SPLINE
SPL {X  -133.736, Y  +773.248, Z    +0.000, E1   -45.385, E3 +353303.340}
SPL {X  -160.761, Y  +715.447, Z    +0.000, E1   -23.748, E3 +353260.190}
SPL {X  -164.304, Y  +696.571, Z    +0.000, E1   -14.525, E3 +353265.413}
SPL {X  -165.498, Y  +682.585, Z    +0.000, E1    -6.769, E3 +353265.088}
SPL {X  -165.650, Y  +674.975, Z    +0.000, E1    -1.888, E3 +353263.446}
SPL {X  -165.650, Y  +671.520, Z    +0.000, E1    +0.682, E3 +353262.373}
SPL {X  -165.650, Y  +668.289, Z    +0.000, E1    +3.417, E3 +353262.215}
SPL {X  -165.650, Y  +663.040, Z    +0.000, E1    +8.602, E3 +353261.410}
SPL {X  -165.650, Y  +655.692, Z    +0.000, E1   +17.061, E3 +353259.945}
SPL {X  -165.650, Y  +646.511, Z    +0.000, E1   +26.434, E3 +353262.725}
SPL {X  -165.650, Y  +637.905, Z    +0.000, E1   +40.225, E3 +353250.850}
SPL {X  -165.650, Y  +611.479, Z    +0.000, E1   +52.226, E3 +353264.402}
SPL {X  -165.650, Y  +599.923, Z    +0.000, E1   +51.240, E3 +353281.492}
SPL {X  -165.650, Y  +553.219, Z    +0.000, E1   +52.865, E3 +353338.252}
ENDSPLINE

SPLINE
SPL {X  -165.650, Y  +569.883, Z    +0.000, E1   +45.183, E3 +353353.929}
ENDSPLINE

SPLINE
SPL {X  -165.650, Y  +561.960, Z    +0.000, E1   +45.285, E3 +353369.584}
SPL {X  -165.650, Y  +554.065, Z    +0.000, E1   +45.254, E3 +353385.646}
SPL {X  -165.650, Y  +548.074, Z    +0.000, E1   +45.245, E3 +353397.757}
SPL {X  -165.650, Y  +542.958, Z    +0.000, E1   +45.131, E3 +353408.888}
SPL {X  -165.650, Y  +535.288, Z    +0.000, E1   +45.332, E3 +353423.328}
SPL {X  -165.650, Y  +529.160, Z    +0.000, E1   +45.215, E3 +353436.309}
SPL {X  -165.650, Y  +522.672, Z    +0.000, E1   +45.331, E3 +353448.876}
SPL {X  -165.650, Y  +516.211, Z    +0.000, E1   +45.175, E3 +353462.835}
SPL {X  -165.650, Y  +509.762, Z    +0.000, E1   +45.191, E3 +353475.877}
SPL {X  -165.650, Y  +503.812, Z    +0.000, E1   +45.188, E3 +353487.916}
SPL {X  -165.650, Y  +499.646, Z    +0.000, E1   +44.886, E3 +353498.187}
ENDSPLINE

SPLINE
SPL {X  -165.650, Y  +514.834, Z    +0.000, E1   +36.829, E3 +353510.953}
ENDSPLINE

SPLINE
SPL {X  -165.650, Y  +506.421, Z    +0.000, E1   +37.886, E3 +353527.065}
SPL {X  -165.650, Y  +499.917, Z    +0.000, E1   +38.752, E3 +353538.526}
SPL {X  -165.650, Y  +493.826, Z    +0.000, E1   +39.521, E3 +353549.280}
SPL {X  -165.650, Y  +487.003, Z    +0.000, E1   +40.380, E3 +353560.734}
SPL {X  -165.650, Y  +478.382, Z    +0.000, E1   +41.628, E3 +353573.647}
SPL {X  -165.650, Y  +472.112, Z    +0.000, E1   +42.202, E3 +353584.386}
SPL {X  -165.650, Y  +466.741, Z    +0.000, E1   +42.890, E3 +353592.306}
SPL {X  -165.650, Y  +458.202, Z    +0.000, E1   +44.020, E3 +353604.094}
SPL {X  -165.650, Y  +449.099, Z    +0.000, E1   +44.871, E3 +353618.056}
SPL {X  -165.650, Y  +442.120, Z    +0.000, E1   +45.313, E3 +353629.608}
SPL {X  -165.650, Y  +436.063, Z    +0.000, E1   +44.972, E3 +353644.193}
SPL {X  -165.650, Y  +427.943, Z    +0.000, E1   +45.362, E3 +353658.230}
SPL {X  -165.650, Y  +422.523, Z    +0.000, E1   +45.103, E3 +353670.908}
SPL {X  -165.650, Y  +415.564, Z    +0.000, E1   +45.195, E3 +353684.447}
SPL {X  -165.650, Y  +410.687, Z    +0.000, E1   +44.955, E3 +353695.763}
SPL {X  -165.650, Y  +405.522, Z    +0.000, E1   +45.119, E3 +353705.324}
SPL {X  -165.650, Y  +399.216, Z    +0.000, E1   +45.246, E3 +353717.517}
SPL {X  -165.650, Y  +391.618, Z    +0.000, E1   +45.037, E3 +353734.296}
SPL {X  -165.650, Y  +383.700, Z    +0.000, E1   +45.345, E3 +353748.422}
SPL {X  -165.650, Y  +379.225, Z    +0.000, E1   +45.073, E3 +353759.111}
SPL {X  -165.591, Y  +374.097, Z    +0.000, E1   +45.069, E3 +353769.592}
SPL {X  -165.372, Y  +368.914, Z    +0.000, E1   +45.103, E3 +353779.952}
SPL {X  -164.987, Y  +363.696, Z    +0.000, E1   +45.006, E3 +353791.175}
SPL {X  -164.256, Y  +357.053, Z    +0.000, E1   +44.969, E3 +353804.978}
SPL {X  -163.441, Y  +351.538, Z    +0.000, E1   +44.749, E3 +353817.341}
SPL {X  -162.419, Y  +345.942, Z    +0.000, E1   +44.540, E3 +353830.073}
SPL {X  -161.210, Y  +340.404, Z    +0.000, E1   +44.250, E3 +353842.898}
SPL {X  -159.961, Y  +335.460, Z    +0.000, E1   +44.205, E3 +353853.261}
SPL {X  -158.595, Y  +330.672, Z    +0.000, E1   +43.797, E3 +353865.239}
SPL {X  -157.207, Y  +326.289, Z    +0.000, E1   +43.631, E3 +353874.992}
SPL {X  -152.192, Y  +313.097, Z    +0.000, E1   +47.715, E3 +353878.546}
SPL {X  -146.385, Y  +300.967, Z    +0.000, E1   +50.402, E3 +353884.741}
SPL {X  -137.641, Y  +286.333, Z    +0.000, E1   +45.396, E3 +353956.232}
SPL {X  -137.518, Y  +286.149, Z    +0.000, E1   +42.648, E3 +354028.741}
ENDSPLINE

SPLINE
SPL {X  -156.430, Y  +324.005, Z    +0.000, E1   +29.926, E3 +354033.876}
SPL {X  -161.387, Y  +341.161, Z    +0.000, E1   +22.590, E3 +354049.718}
SPL {X  -164.566, Y  +359.576, Z    +0.000, E1   +13.425, E3 +354028.311}
SPL {X  -165.355, Y  +368.611, Z    +0.000, E1    +8.407, E3 +354031.892}
SPL {X  -165.614, Y  +375.050, Z    +0.000, E1    +4.520, E3 +354033.196}
SPL {X  -165.650, Y  +379.847, Z    +0.000, E1    +1.364, E3 +354031.545}
SPL {X  -165.650, Y  +384.387, Z    +0.000, E1    -2.084, E3 +354030.527}
SPL {X  -165.650, Y  +387.977, Z    +0.000, E1    -5.454, E3 +354031.012}
SPL {X  -165.650, Y  +392.464, Z    +0.000, E1   -10.170, E3 +354028.695}
SPL {X  -165.650, Y  +397.361, Z    +0.000, E1   -15.736, E3 +354028.027}
SPL {X  -165.650, Y  +404.553, Z    +0.000, E1   -23.488, E3 +354028.803}
SPL {X  -165.650, Y  +415.773, Z    +0.000, E1   -36.308, E3 +354024.955}
SPL {X  -165.650, Y  +461.620, Z    +0.000, E1   -55.594, E3 +354044.685}
SPL {X  -165.650, Y  +498.574, Z    +0.000, E1   -52.082, E3 +354105.710}
ENDSPLINE

SPLINE
SPL {X  -165.650, Y  +484.983, Z    +0.000, E1   -45.406, E3 +354121.213}
ENDSPLINE

SPLINE
SPL {X  -165.650, Y  +492.090, Z    +0.000, E1   -45.292, E3 +354136.235}
SPL {X  -165.650, Y  +498.857, Z    +0.000, E1   -45.339, E3 +354149.572}
SPL {X  -165.650, Y  +505.115, Z    +0.000, E1   -45.299, E3 +354162.520}
SPL {X  -165.650, Y  +510.931, Z    +0.000, E1   -45.250, E3 +354174.511}
SPL {X  -165.650, Y  +516.157, Z    +0.000, E1   -45.240, E3 +354185.186}
SPL {X  -165.650, Y  +521.049, Z    +0.000, E1   -45.236, E3 +354195.138}
SPL {X  -165.650, Y  +527.050, Z    +0.000, E1   -45.345, E3 +354206.634}
SPL {X  -165.650, Y  +532.042, Z    +0.000, E1   -45.233, E3 +354217.378}
SPL {X  -165.650, Y  +537.290, Z    +0.000, E1   -45.204, E3 +354228.219}
SPL {X  -165.650, Y  +544.196, Z    +0.000, E1   -45.432, E3 +354240.893}
SPL {X  -165.650, Y  +548.678, Z    +0.000, E1   -45.162, E3 +354251.457}
SPL {X  -165.650, Y  +554.600, Z    +0.000, E1   -45.345, E3 +354262.434}
SPL {X  -165.650, Y  +559.896, Z    +0.000, E1   -45.150, E3 +354274.289}
SPL {X  -165.650, Y  +566.830, Z    +0.000, E1   -45.346, E3 +354287.269}
SPL {X  -165.650, Y  +573.074, Z    +0.000, E1   -45.379, E3 +354299.600}
SPL {X  -165.650, Y  +579.360, Z    +0.000, E1   -45.300, E3 +354312.885}
SPL {X  -165.650, Y  +584.577, Z    +0.000, E1   -45.167, E3 +354324.108}
SPL {X  -165.650, Y  +590.060, Z    +0.000, E1   -45.221, E3 +354334.999}
SPL {X  -165.650, Y  +596.611, Z    +0.000, E1   -45.390, E3 +354347.236}
SPL {X  -165.650, Y  +603.637, Z    +0.000, E1   -45.296, E3 +354362.154}
SPL {X  -165.650, Y  +610.850, Z    +0.000, E1   -45.208, E3 +354377.162}
SPL {X  -165.650, Y  +617.450, Z    +0.000, E1   -45.402, E3 +354389.365}
SPL {X  -165.650, Y  +622.720, Z    +0.000, E1   -45.272, E3 +354400.763}
SPL {X  -165.650, Y  +627.828, Z    +0.000, E1   -45.174, E3 +354411.719}
SPL {X  -165.650, Y  +634.620, Z    +0.000, E1   -45.438, E3 +354423.925}
SPL {X  -165.650, Y  +640.808, Z    +0.000, E1   -45.294, E3 +354437.299}
SPL {X  -165.650, Y  +646.552, Z    +0.000, E1   -45.137, E3 +354449.824}
SPL {X  -165.650, Y  +652.431, Z    +0.000, E1   -45.333, E3 +354460.578}
SPL {X  -165.650, Y  +657.443, Z    +0.000, E1   -45.316, E3 +354470.834}
SPL {X  -165.650, Y  +662.999, Z    +0.000, E1   -45.214, E3 +354482.706}
SPL {X  -165.650, Y  +668.737, Z    +0.000, E1   -45.236, E3 +354494.221}
SPL {X  -165.650, Y  +675.226, Z    +0.000, E1   -45.503, E3 +354505.725}
SPL {X  -165.597, Y  +679.672, Z    +0.000, E1   -45.206, E3 +354516.446}
SPL {X  -165.388, Y  +684.808, Z    +0.000, E1   -45.192, E3 +354526.954}
SPL {X  -165.020, Y  +689.938, Z    +0.000, E1   -45.107, E3 +354537.896}
SPL {X  -164.358, Y  +696.147, Z    +0.000, E1   -45.160, E3 +354550.162}
SPL {X  -163.631, Y  +701.286, Z    +0.000, E1   -44.994, E3 +354561.454}
SPL {X  -162.679, Y  +706.734, Z    +0.000, E1   -44.812, E3 +354573.687}
SPL {X  -161.655, Y  +711.661, Z    +0.000, E1   -44.525, E3 +354585.068}
SPL {X  -160.692, Y  +715.726, Z    +0.000, E1   -44.379, E3 +354594.225}
SPL {X  -159.384, Y  +720.631, Z    +0.000, E1   -44.155, E3 +354605.376}
SPL {X  -158.321, Y  +724.227, Z    +0.000, E1   -43.955, E3 +354613.697}
SPL {X  -156.604, Y  +729.490, Z    +0.000, E1   -44.229, E3 +354622.863}
SPL {X  -147.100, Y  +751.668, Z    +0.000, E1   -50.624, E3 +354628.750}
SPL {X  -144.116, Y  +757.172, Z    +0.000, E1   -42.809, E3 +354698.146}
SPL {X  -127.227, Y  +781.582, Z    +0.000, E1   -46.780, E3 +354743.816}
ENDSPLINE

SPLINE
SPL {X  -133.736, Y  +773.248, Z    +0.000, E1   -45.385, E3 +354821.858}
SPL {X  -160.761, Y  +715.447, Z    +0.000, E1   -23.748, E3 +354778.708}
SPL {X  -164.304, Y  +696.571, Z    +0.000, E1   -14.525, E3 +354783.932}
SPL {X  -165.498, Y  +682.585, Z    +0.000, E1    -6.769, E3 +354783.606}
SPL {X  -165.650, Y  +674.975, Z    +0.000, E1    -1.888, E3 +354781.965}
SPL {X  -165.650, Y  +671.520, Z    +0.000, E1    +0.682, E3 +354780.892}
SPL {X  -165.650, Y  +668.289, Z    +0.000, E1    +3.417, E3 +354780.734}
SPL {X  -165.650, Y  +663.040, Z    +0.000, E1    +8.602, E3 +354779.928}
SPL {X  -165.650, Y  +655.692, Z    +0.000, E1   +17.061, E3 +354778.464}
SPL {X  -165.650, Y  +646.511, Z    +0.000, E1   +26.434, E3 +354781.244}
SPL {X  -165.650, Y  +637.905, Z    +0.000, E1   +40.225, E3 +354769.368}
SPL {X  -165.650, Y  +611.479, Z    +0.000, E1   +52.226, E3 +354782.921}
SPL {X  -165.650, Y  +599.923, Z    +0.000, E1   +51.240, E3 +354800.010}
SPL {X  -165.650, Y  +553.219, Z    +0.000, E1   +52.865, E3 +354856.771}
ENDSPLINE

SPLINE
SPL {X  -165.650, Y  +569.883, Z    +0.000, E1   +45.183, E3 +354872.447}
ENDSPLINE

SPLINE
SPL {X  -165.650, Y  +561.960, Z    +0.000, E1   +45.285, E3 +354888.103}
SPL {X  -165.650, Y  +554.065, Z    +0.000, E1   +45.254, E3 +354904.165}
SPL {X  -165.650, Y  +548.074, Z    +0.000, E1   +45.245, E3 +354916.275}
SPL {X  -165.650, Y  +542.958, Z    +0.000, E1   +45.131, E3 +354927.406}
SPL {X  -165.650, Y  +535.288, Z    +0.000, E1   +45.332, E3 +354941.847}
SPL {X  -165.650, Y  +529.160, Z    +0.000, E1   +45.215, E3 +354954.828}
SPL {X  -165.650, Y  +522.672, Z    +0.000, E1   +45.331, E3 +354967.394}
SPL {X  -165.650, Y  +516.211, Z    +0.000, E1   +45.175, E3 +354981.354}
SPL {X  -165.650, Y  +509.762, Z    +0.000, E1   +45.191, E3 +354994.396}
SPL {X  -165.650, Y  +503.812, Z    +0.000, E1   +45.188, E3 +355006.434}
SPL {X  -165.650, Y  +499.646, Z    +0.000, E1   +44.886, E3 +355016.705}
ENDSPLINE

SPLINE
SPL {X  -165.650, Y  +516.930, Z    +0.000, E1   +36.544, E3 +355025.376}
ENDSPLINE

SPLINE
SPL {X  -165.650, Y  +511.324, Z    +0.000, E1   +37.254, E3 +355036.367}
SPL {X  -165.650, Y  +504.742, Z    +0.000, E1   +38.087, E3 +355048.672}
SPL {X  -165.650, Y  +497.845, Z    +0.000, E1   +39.022, E3 +355060.747}
SPL {X  -165.650, Y  +491.819, Z    +0.000, E1   +39.756, E3 +355071.266}
SPL {X  -165.650, Y  +485.086, Z    +0.000, E1   +40.678, E3 +355082.110}
SPL {X  -165.650, Y  +476.633, Z    +0.000, E1   +41.847, E3 +355094.809}
SPL {X  -165.650, Y  +468.596, Z    +0.000, E1   +42.673, E3 +355108.072}
SPL {X  -165.650, Y  +460.562, Z    +0.000, E1   +43.733, E3 +355119.224}
SPL {X  -165.650, Y  +455.629, Z    +0.000, E1   +44.293, E3 +355126.343}
SPL {X  -165.650, Y  +449.099, Z    +0.000, E1   +44.871, E3 +355136.575}
SPL {X  -165.650, Y  +442.120, Z    +0.000, E1   +45.313, E3 +355148.127}
SPL {X  -165.650, Y  +439.103, Z    +0.000, E1   +44.726, E3 +355157.736}
SPL {X  -165.650, Y  +433.421, Z    +0.000, E1   +45.110, E3 +355167.123}
SPL {X  -165.650, Y  +426.476, Z    +0.000, E1   +45.244, E3 +355180.627}
SPL {X  -165.650, Y  +420.418, Z    +0.000, E1   +45.128, E3 +355193.421}
SPL {X  -165.650, Y  +415.564, Z    +0.000, E1   +45.195, E3 +355202.966}
SPL {X  -165.650, Y  +410.687, Z    +0.000, E1   +44.955, E3 +355214.282}
SPL {X  -165.650, Y  +405.522, Z    +0.000, E1   +45.119, E3 +355223.842}
SPL {X  -165.650, Y  +400.300, Z    +0.000, E1   +45.439, E3 +355232.526}
SPL {X  -165.650, Y  +396.171, Z    +0.000, E1   +44.969, E3 +355243.783}
SPL {X  -165.650, Y  +390.060, Z    +0.000, E1   +45.007, E3 +355256.017}
SPL {X  -165.650, Y  +383.700, Z    +0.000, E1   +45.345, E3 +355266.941}
SPL {X  -165.650, Y  +379.225, Z    +0.000, E1   +45.073, E3 +355277.630}
SPL {X  -165.591, Y  +374.097, Z    +0.000, E1   +45.069, E3 +355288.111}
SPL {X  -165.372, Y  +368.914, Z    +0.000, E1   +45.103, E3 +355298.471}
SPL {X  -164.987, Y  +363.696, Z    +0.000, E1   +45.006, E3 +355309.694}
SPL {X  -164.256, Y  +357.053, Z    +0.000, E1   +44.969, E3 +355323.496}
SPL {X  -163.441, Y  +351.538, Z    +0.000, E1   +44.749, E3 +355335.860}
SPL {X  -162.419, Y  +345.942, Z    +0.000, E1   +44.540, E3 +355348.592}
SPL {X  -161.210, Y  +340.404, Z    +0.000, E1   +44.250, E3 +355361.417}
SPL {X  -159.961, Y  +335.460, Z    +0.000, E1   +44.205, E3 +355371.779}
SPL {X  -158.595, Y  +330.672, Z    +0.000, E1   +43.797, E3 +355383.758}
SPL {X  -157.207, Y  +326.289, Z    +0.000, E1   +43.631, E3 +355393.511}
SPL {X  -152.192, Y  +313.097, Z    +0.000, E1   +47.715, E3 +355397.064}
SPL {X  -146.385, Y  +300.967, Z    +0.000, E1   +50.402, E3 +355403.260}
SPL {X  -138.435, Y  +287.529, Z    +0.000, E1   +45.834, E3 +355465.216}
SPL {X  -134.645, Y  +282.008, Z    +0.000, E1   +45.207, E3 +355494.872}
ENDSPLINE

SPLINE
SPL {X  -154.915, Y  +319.839, Z    +0.000, E1   +31.584, E3 +355554.391}
SPL {X  -161.387, Y  +341.161, Z    +0.000, E1   +22.590, E3 +355568.236}
SPL {X  -164.566, Y  +359.576, Z    +0.000, E1   +13.425, E3 +355546.830}
SPL {X  -165.355, Y  +368.611, Z    +0.000, E1    +8.407, E3 +355550.411}
SPL {X  -165.614, Y  +375.050, Z    +0.000, E1    +4.520, E3 +355551.714}
SPL {X  -165.650, Y  +379.847, Z    +0.000, E1    +1.364, E3 +355550.064}
SPL {X  -165.650, Y  +383.246, Z    +0.000, E1    -1.216, E3 +355549.157}
SPL {X  -165.650, Y  +386.866, Z    +0.000, E1    -4.337, E3 +355549.210}
SPL {X  -165.650, Y  +392.464, Z    +0.000, E1   -10.170, E3 +355547.213}
SPL {X  -165.650, Y  +397.361, Z    +0.000, E1   -15.736, E3 +355546.545}
SPL {X  -165.650, Y  +404.553, Z    +0.000, E1   -23.488, E3 +355547.321}
SPL {X  -165.650, Y  +415.773, Z    +0.000, E1   -36.308, E3 +355543.474}
SPL {X  -165.650, Y  +456.525, Z    +0.000, E1   -55.091, E3 +355559.036}
SPL {X  -165.650, Y  +467.178, Z    +0.000, E1   -56.049, E3 +355567.773}
SPL {X  -165.650, Y  +498.574, Z    +0.000, E1   -52.082, E3 +355624.228}
ENDSPLINE

SPLINE
SPL {X  -165.650, Y  +484.983, Z    +0.000, E1   -45.406, E3 +355639.731}
ENDSPLINE

SPLINE
SPL {X  -165.650, Y  +492.090, Z    +0.000, E1   -45.292, E3 +355654.754}
SPL {X  -165.650, Y  +498.857, Z    +0.000, E1   -45.339, E3 +355668.091}
SPL {X  -165.650, Y  +504.159, Z    +0.000, E1   -45.384, E3 +355678.485}
SPL {X  -165.650, Y  +509.628, Z    +0.000, E1   -45.217, E3 +355690.669}
SPL {X  -165.650, Y  +516.157, Z    +0.000, E1   -45.240, E3 +355703.704}
SPL {X  -165.650, Y  +521.049, Z    +0.000, E1   -45.236, E3 +355713.657}
SPL {X  -165.650, Y  +527.050, Z    +0.000, E1   -45.345, E3 +355725.153}
SPL {X  -165.650, Y  +532.042, Z    +0.000, E1   -45.233, E3 +355735.896}
SPL {X  -165.650, Y  +537.290, Z    +0.000, E1   -45.204, E3 +355746.737}
SPL {X  -165.650, Y  +544.196, Z    +0.000, E1   -45.432, E3 +355759.411}
SPL {X  -165.650, Y  +548.678, Z    +0.000, E1   -45.162, E3 +355769.975}
SPL {X  -165.650, Y  +554.600, Z    +0.000, E1   -45.345, E3 +355780.952}
SPL {X  -165.650, Y  +561.799, Z    +0.000, E1   -45.312, E3 +355795.821}
SPL {X  -165.650, Y  +567.835, Z    +0.000, E1   -45.186, E3 +355808.628}
SPL {X  -165.650, Y  +573.074, Z    +0.000, E1   -45.379, E3 +355818.118}
SPL {X  -165.650, Y  +577.292, Z    +0.000, E1   -45.246, E3 +355827.382}
SPL {X  -165.650, Y  +583.131, Z    +0.000, E1   -45.255, E3 +355839.324}
SPL {X  -165.650, Y  +590.060, Z    +0.000, E1   -45.221, E3 +355853.518}
SPL {X  -165.650, Y  +596.611, Z    +0.000, E1   -45.390, E3 +355865.754}
SPL {X  -165.650, Y  +603.637, Z    +0.000, E1   -45.296, E3 +355880.673}
SPL {X  -165.650, Y  +610.850, Z    +0.000, E1   -45.208, E3 +355895.681}
SPL {X  -165.650, Y  +617.450, Z    +0.000, E1   -45.402, E3 +355907.883}
SPL {X  -165.650, Y  +622.720, Z    +0.000, E1   -45.272, E3 +355919.281}
SPL {X  -165.650, Y  +627.828, Z    +0.000, E1   -45.174, E3 +355930.238}
SPL {X  -165.650, Y  +634.620, Z    +0.000, E1   -45.438, E3 +355942.443}
SPL {X  -165.650, Y  +640.808, Z    +0.000, E1   -45.294, E3 +355955.818}
SPL {X  -165.650, Y  +646.552, Z    +0.000, E1   -45.137, E3 +355968.342}
SPL {X  -165.650, Y  +652.431, Z    +0.000, E1   -45.333, E3 +355979.097}
SPL {X  -165.650, Y  +657.443, Z    +0.000, E1   -45.316, E3 +355989.353}
SPL {X  -165.650, Y  +662.999, Z    +0.000, E1   -45.214, E3 +356001.225}
SPL {X  -165.650, Y  +668.737, Z    +0.000, E1   -45.236, E3 +356012.740}
SPL {X  -165.650, Y  +675.226, Z    +0.000, E1   -45.503, E3 +356024.243}
SPL {X  -165.597, Y  +679.672, Z    +0.000, E1   -45.206, E3 +356034.965}
SPL {X  -165.388, Y  +684.808, Z    +0.000, E1   -45.192, E3 +356045.472}
SPL {X  -165.020, Y  +689.938, Z    +0.000, E1   -45.107, E3 +356056.415}
SPL {X  -164.358, Y  +696.147, Z    +0.000, E1   -45.160, E3 +356068.681}
SPL {X  -163.631, Y  +701.286, Z    +0.000, E1   -44.994, E3 +356079.973}
SPL {X  -163.047, Y  +704.748, Z    +0.000, E1   -44.682, E3 +356088.796}
SPL {X  -161.884, Y  +710.619, Z    +0.000, E1   -44.738, E3 +356100.421}
SPL {X  -160.692, Y  +715.726, Z    +0.000, E1   -44.379, E3 +356112.744}
SPL {X  -158.938, Y  +722.175, Z    +0.000, E1   -44.121, E3 +356127.392}
SPL {X  -157.296, Y  +727.442, Z    +0.000, E1   -43.792, E3 +356139.617}
SPL {X  -153.030, Y  +738.918, Z    +0.000, E1   -47.123, E3 +356143.983}
SPL {X  -145.149, Y  +755.323, Z    +0.000, E1   -51.167, E3 +356150.115}
SPL {X  -143.038, Y  +759.047, Z    +0.000, E1   -43.157, E3 +356219.289}
SPL {X  -123.277, Y  +786.146, Z    +0.000, E1   -47.533, E3 +356275.344}
ENDSPLINE

SPLINE
SPL {X  -133.736, Y  +773.248, Z    +0.000, E1   -45.385, E3 +356340.377}
SPL {X  -160.761, Y  +715.447, Z    +0.000, E1   -23.748, E3 +356297.227}
SPL {X  -164.304, Y  +696.571, Z    +0.000, E1   -14.525, E3 +356302.451}
SPL {X  -165.498, Y  +682.585, Z    +0.000, E1    -6.769, E3 +356302.125}
SPL {X  -165.650, Y  +674.975, Z    +0.000, E1    -1.888, E3 +356300.483}
SPL {X  -165.650, Y  +671.520, Z    +0.000, E1    +0.682, E3 +356299.410}
SPL {X  -165.650, Y  +668.289, Z    +0.000, E1    +3.417, E3 +356299.252}
SPL {X  -165.650, Y  +663.040, Z    +0.000, E1    +8.602, E3 +356298.447}
SPL {X  -165.650, Y  +655.692, Z    +0.000, E1   +17.061, E3 +356296.982}
SPL {X  -165.650, Y  +646.511, Z    +0.000, E1   +26.434, E3 +356299.762}
SPL {X  -165.650, Y  +637.905, Z    +0.000, E1   +40.225, E3 +356287.887}
SPL {X  -165.650, Y  +611.479, Z    +0.000, E1   +52.226, E3 +356301.439}
SPL {X  -165.650, Y  +599.923, Z    +0.000, E1   +51.240, E3 +356318.529}
SPL {X  -165.650, Y  +553.219, Z    +0.000, E1   +52.865, E3 +356375.289}
ENDSPLINE

SPLINE
SPL {X  -165.650, Y  +569.883, Z    +0.000, E1   +45.183, E3 +356390.966}
ENDSPLINE

SPLINE
SPL {X  -165.650, Y  +561.960, Z    +0.000, E1   +45.285, E3 +356406.621}
SPL {X  -165.650, Y  +554.065, Z    +0.000, E1   +45.254, E3 +356422.683}
SPL {X  -165.650, Y  +548.074, Z    +0.000, E1   +45.245, E3 +356434.794}
SPL {X  -165.650, Y  +542.958, Z    +0.000, E1   +45.131, E3 +356445.925}
SPL {X  -165.650, Y  +535.288, Z    +0.000, E1   +45.332, E3 +356460.366}
SPL {X  -165.650, Y  +529.160, Z    +0.000, E1   +45.215, E3 +356473.346}
SPL {X  -165.650, Y  +522.672, Z    +0.000, E1   +45.331, E3 +356485.913}
SPL {X  -165.650, Y  +516.211, Z    +0.000, E1   +45.175, E3 +356499.872}
SPL {X  -165.650, Y  +509.762, Z    +0.000, E1   +45.191, E3 +356512.914}
SPL {X  -165.650, Y  +503.812, Z    +0.000, E1   +45.188, E3 +356524.953}
SPL {X  -165.650, Y  +499.646, Z    +0.000, E1   +44.886, E3 +356535.224}
ENDSPLINE

SPLINE
SPL {X  -165.650, Y  +514.834, Z    +0.000, E1   +36.829, E3 +356547.990}
ENDSPLINE

SPLINE
SPL {X  -165.650, Y  +506.421, Z    +0.000, E1   +37.886, E3 +356564.102}
SPL {X  -165.650, Y  +499.917, Z    +0.000, E1   +38.752, E3 +356575.563}
SPL {X  -165.650, Y  +493.826, Z    +0.000, E1   +39.521, E3 +356586.317}
SPL {X  -165.650, Y  +487.003, Z    +0.000, E1   +40.380, E3 +356597.771}
SPL {X  -165.650, Y  +478.382, Z    +0.000, E1   +41.628, E3 +356610.684}
SPL {X  -165.650, Y  +472.112, Z    +0.000, E1   +42.202, E3 +356621.423}
SPL {X  -165.650, Y  +466.741, Z    +0.000, E1   +42.890, E3 +356629.343}
SPL {X  -165.650, Y  +458.202, Z    +0.000, E1   +44.020, E3 +356641.131}
SPL {X  -165.650, Y  +449.099, Z    +0.000, E1   +44.871, E3 +356655.093}
SPL {X  -165.650, Y  +442.120, Z    +0.000, E1   +45.313, E3 +356666.645}
SPL {X  -165.650, Y  +436.063, Z    +0.000, E1   +44.972, E3 +356681.230}
SPL {X  -165.650, Y  +427.943, Z    +0.000, E1   +45.362, E3 +356695.267}
SPL {X  -165.650, Y  +422.523, Z    +0.000, E1   +45.103, E3 +356707.945}
SPL {X  -165.650, Y  +415.564, Z    +0.000, E1   +45.195, E3 +356721.484}
SPL {X  -165.650, Y  +410.687, Z    +0.000, E1   +44.955, E3 +356732.801}
SPL {X  -165.650, Y  +405.522, Z    +0.000, E1   +45.119, E3 +356742.361}
SPL {X  -165.650, Y  +399.216, Z    +0.000, E1   +45.246, E3 +356754.555}
SPL {X  -165.650, Y  +391.618, Z    +0.000, E1   +45.037, E3 +356771.333}
SPL {X  -165.650, Y  +383.700, Z    +0.000, E1   +45.345, E3 +356785.459}
SPL {X  -165.650, Y  +379.225, Z    +0.000, E1   +45.073, E3 +356796.148}
SPL {X  -165.591, Y  +374.097, Z    +0.000, E1   +45.069, E3 +356806.629}
SPL {X  -165.372, Y  +368.914, Z    +0.000, E1   +45.103, E3 +356816.989}
SPL {X  -164.987, Y  +363.696, Z    +0.000, E1   +45.006, E3 +356828.212}
SPL {X  -164.256, Y  +357.053, Z    +0.000, E1   +44.969, E3 +356842.015}
SPL {X  -163.441, Y  +351.538, Z    +0.000, E1   +44.749, E3 +356854.378}
SPL {X  -162.419, Y  +345.942, Z    +0.000, E1   +44.540, E3 +356867.110}
SPL {X  -161.210, Y  +340.404, Z    +0.000, E1   +44.250, E3 +356879.935}
SPL {X  -159.961, Y  +335.460, Z    +0.000, E1   +44.205, E3 +356890.298}
SPL {X  -158.595, Y  +330.672, Z    +0.000, E1   +43.797, E3 +356902.276}
SPL {X  -157.207, Y  +326.289, Z    +0.000, E1   +43.631, E3 +356912.029}
SPL {X  -152.192, Y  +313.097, Z    +0.000, E1   +47.715, E3 +356915.583}
SPL {X  -146.385, Y  +300.967, Z    +0.000, E1   +50.402, E3 +356921.778}
SPL {X  -137.641, Y  +286.333, Z    +0.000, E1   +45.396, E3 +356993.269}
SPL {X  -137.518, Y  +286.149, Z    +0.000, E1   +42.648, E3 +357065.779}
ENDSPLINE

SPLINE
SPL {X  -156.430, Y  +324.005, Z    +0.000, E1   +29.926, E3 +357070.913}
SPL {X  -161.387, Y  +341.161, Z    +0.000, E1   +22.590, E3 +357086.755}
SPL {X  -164.566, Y  +359.576, Z    +0.000, E1   +13.425, E3 +357065.348}
SPL {X  -165.355, Y  +368.611, Z    +0.000, E1    +8.407, E3 +357068.929}
SPL {X  -165.614, Y  +375.050, Z    +0.000, E1    +4.520, E3 +357070.233}
SPL {X  -165.650, Y  +379.847, Z    +0.000, E1    +1.364, E3 +357068.582}
SPL {X  -165.650, Y  +384.387, Z    +0.000, E1    -2.084, E3 +357067.564}
SPL {X  -165.650, Y  +387.977, Z    +0.000, E1    -5.454, E3 +357068.049}
SPL {X  -165.650, Y  +392.464, Z    +0.000, E1   -10.170, E3 +357065.732}
SPL {X  -165.650, Y  +397.361, Z    +0.000, E1   -15.736, E3 +357065.064}
SPL {X  -165.650, Y  +404.553, Z    +0.000, E1   -23.488, E3 +357065.840}
SPL {X  -165.650, Y  +415.773, Z    +0.000, E1   -36.308, E3 +357061.992}
SPL {X  -165.650, Y  +461.620, Z    +0.000, E1   -55.594, E3 +357081.722}
SPL {X  -165.650, Y  +498.574, Z    +0.000, E1   -52.082, E3 +357142.747}
ENDSPLINE

SPLINE
SPL {X  -165.650, Y  +484.983, Z    +0.000, E1   -45.406, E3 +357158.250}
ENDSPLINE

SPLINE
SPL {X  -165.650, Y  +492.090, Z    +0.000, E1   -45.292, E3 +357173.272}
SPL {X  -165.650, Y  +498.857, Z    +0.000, E1   -45.339, E3 +357186.609}
SPL {X  -165.650, Y  +505.115, Z    +0.000, E1   -45.299, E3 +357199.558}
SPL {X  -165.650, Y  +510.931, Z    +0.000, E1   -45.250, E3 +357211.548}
SPL {X  -165.650, Y  +516.157, Z    +0.000, E1   -45.240, E3 +357222.223}
SPL {X  -165.650, Y  +521.049, Z    +0.000, E1   -45.236, E3 +357232.175}
SPL {X  -165.650, Y  +527.050, Z    +0.000, E1   -45.345, E3 +357243.671}
SPL {X  -165.650, Y  +532.042, Z    +0.000, E1   -45.233, E3 +357254.415}
SPL {X  -165.650, Y  +537.290, Z    +0.000, E1   -45.204, E3 +357265.256}
SPL {X  -165.650, Y  +544.196, Z    +0.000, E1   -45.432, E3 +357277.930}
SPL {X  -165.650, Y  +548.678, Z    +0.000, E1   -45.162, E3 +357288.494}
SPL {X  -165.650, Y  +554.600, Z    +0.000, E1   -45.345, E3 +357299.471}
SPL {X  -165.650, Y  +559.896, Z    +0.000, E1   -45.150, E3 +357311.326}
SPL {X  -165.650, Y  +566.830, Z    +0.000, E1   -45.346, E3 +357324.306}
SPL {X  -165.650, Y  +573.074, Z    +0.000, E1   -45.379, E3 +357336.637}
SPL {X  -165.650, Y  +579.360, Z    +0.000, E1   -45.300, E3 +357349.922}
SPL {X  -165.650, Y  +584.577, Z    +0.000, E1   -45.167, E3 +357361.145}
SPL {X  -165.650, Y  +590.060, Z    +0.000, E1   -45.221, E3 +357372.036}
SPL {X  -165.650, Y  +596.611, Z    +0.000, E1   -45.390, E3 +357384.273}
SPL {X  -165.650, Y  +603.637, Z    +0.000, E1   -45.296, E3 +357399.191}
SPL {X  -165.650, Y  +610.850, Z    +0.000, E1   -45.208, E3 +357414.199}
SPL {X  -165.650, Y  +617.450, Z    +0.000, E1   -45.402, E3 +357426.402}
SPL {X  -165.650, Y  +622.720, Z    +0.000, E1   -45.272, E3 +357437.800}
SPL {X  -165.650, Y  +627.828, Z    +0.000, E1   -45.174, E3 +357448.756}
SPL {X  -165.650, Y  +634.620, Z    +0.000, E1   -45.438, E3 +357460.962}
SPL {X  -165.650, Y  +640.808, Z    +0.000, E1   -45.294, E3 +357474.336}
SPL {X  -165.650, Y  +646.552, Z    +0.000, E1   -45.137, E3 +357486.861}
SPL {X  -165.650, Y  +652.431, Z    +0.000, E1   -45.333, E3 +357497.615}
SPL {X  -165.650, Y  +657.443, Z    +0.000, E1   -45.316, E3 +357507.871}
SPL {X  -165.650, Y  +662.999, Z    +0.000, E1   -45.214, E3 +357519.743}
SPL {X  -165.650, Y  +668.737, Z    +0.000, E1   -45.236, E3 +357531.258}
SPL {X  -165.650, Y  +675.226, Z    +0.000, E1   -45.503, E3 +357542.762}
SPL {X  -165.597, Y  +679.672, Z    +0.000, E1   -45.206, E3 +357553.483}
SPL {X  -165.388, Y  +684.808, Z    +0.000, E1   -45.192, E3 +357563.991}
SPL {X  -165.020, Y  +689.938, Z    +0.000, E1   -45.107, E3 +357574.933}
SPL {X  -164.358, Y  +696.147, Z    +0.000, E1   -45.160, E3 +357587.199}
SPL {X  -163.631, Y  +701.286, Z    +0.000, E1   -44.994, E3 +357598.491}
SPL {X  -162.679, Y  +706.734, Z    +0.000, E1   -44.812, E3 +357610.724}
SPL {X  -161.655, Y  +711.661, Z    +0.000, E1   -44.525, E3 +357622.105}
SPL {X  -160.692, Y  +715.726, Z    +0.000, E1   -44.379, E3 +357631.262}
SPL {X  -159.384, Y  +720.631, Z    +0.000, E1   -44.155, E3 +357642.413}
SPL {X  -158.321, Y  +724.227, Z    +0.000, E1   -43.955, E3 +357650.734}
SPL {X  -156.604, Y  +729.490, Z    +0.000, E1   -44.229, E3 +357659.900}
SPL {X  -147.100, Y  +751.668, Z    +0.000, E1   -50.624, E3 +357665.787}
SPL {X  -144.116, Y  +757.172, Z    +0.000, E1   -42.809, E3 +357735.183}
SPL {X  -127.227, Y  +781.582, Z    +0.000, E1   -46.780, E3 +357780.853}
ENDSPLINE

SPLINE
SPL {X  -133.736, Y  +773.248, Z    +0.000, E1   -45.385, E3 +357858.895}
SPL {X  -160.761, Y  +715.447, Z    +0.000, E1   -23.748, E3 +357815.745}
SPL {X  -164.304, Y  +696.571, Z    +0.000, E1   -14.525, E3 +357820.969}
SPL {X  -165.498, Y  +682.585, Z    +0.000, E1    -6.769, E3 +357820.643}
SPL {X  -165.650, Y  +674.975, Z    +0.000, E1    -1.888, E3 +357819.002}
SPL {X  -165.650, Y  +671.520, Z    +0.000, E1    +0.682, E3 +357817.929}
SPL {X  -165.650, Y  +668.289, Z    +0.000, E1    +3.417, E3 +357817.771}
SPL {X  -165.650, Y  +663.040, Z    +0.000, E1    +8.602, E3 +357816.965}
SPL {X  -165.650, Y  +655.692, Z    +0.000, E1   +17.061, E3 +357815.501}
SPL {X  -165.650, Y  +646.511, Z    +0.000, E1   +26.434, E3 +357818.281}
SPL {X  -165.650, Y  +637.905, Z    +0.000, E1   +40.225, E3 +357806.405}
SPL {X  -165.650, Y  +611.479, Z    +0.000, E1   +52.226, E3 +357819.958}
SPL {X  -165.650, Y  +599.923, Z    +0.000, E1   +51.240, E3 +357837.047}
SPL {X  -165.650, Y  +553.219, Z    +0.000, E1   +52.865, E3 +357893.808}
ENDSPLINE

SPLINE
SPL {X  -165.650, Y  +569.883, Z    +0.000, E1   +45.183, E3 +357909.484}
ENDSPLINE

SPLINE
SPL {X  -165.650, Y  +561.960, Z    +0.000, E1   +45.285, E3 +357925.140}
SPL {X  -165.650, Y  +554.065, Z    +0.000, E1   +45.254, E3 +357941.202}
SPL {X  -165.650, Y  +548.074, Z    +0.000, E1   +45.245, E3 +357953.312}
SPL {X  -165.650, Y  +542.958, Z    +0.000, E1   +45.131, E3 +357964.443}
SPL {X  -165.650, Y  +535.288, Z    +0.000, E1   +45.332, E3 +357978.884}
SPL {X  -165.650, Y  +529.160, Z    +0.000, E1   +45.215, E3 +357991.865}
SPL {X  -165.650, Y  +522.672, Z    +0.000, E1   +45.331, E3 +358004.431}
SPL {X  -165.650, Y  +516.211, Z    +0.000, E1   +45.175, E3 +358018.391}
SPL {X  -165.650, Y  +509.762, Z    +0.000, E1   +45.191, E3 +358031.433}
SPL {X  -165.650, Y  +503.812, Z    +0.000, E1   +45.188, E3 +358043.471}
SPL {X  -165.650, Y  +499.646, Z    +0.000, E1   +44.886, E3 +358053.743}
ENDSPLINE

SPLINE
SPL {X  -165.650, Y  +516.930, Z    +0.000, E1   +36.544, E3 +358062.413}
ENDSPLINE

SPLINE
SPL {X  -165.650, Y  +511.324, Z    +0.000, E1   +37.254, E3 +358073.404}
SPL {X  -165.650, Y  +504.742, Z    +0.000, E1   +38.087, E3 +358085.709}
SPL {X  -165.650, Y  +497.845, Z    +0.000, E1   +39.022, E3 +358097.784}
SPL {X  -165.650, Y  +491.819, Z    +0.000, E1   +39.756, E3 +358108.303}
SPL {X  -165.650, Y  +485.086, Z    +0.000, E1   +40.678, E3 +358119.147}
SPL {X  -165.650, Y  +476.633, Z    +0.000, E1   +41.847, E3 +358131.846}
SPL {X  -165.650, Y  +468.596, Z    +0.000, E1   +42.673, E3 +358145.109}
SPL {X  -165.650, Y  +460.562, Z    +0.000, E1   +43.733, E3 +358156.261}
SPL {X  -165.650, Y  +455.629, Z    +0.000, E1   +44.293, E3 +358163.380}
SPL {X  -165.650, Y  +449.099, Z    +0.000, E1   +44.871, E3 +358173.612}
SPL {X  -165.650, Y  +442.120, Z    +0.000, E1   +45.313, E3 +358185.164}
SPL {X  -165.650, Y  +439.103, Z    +0.000, E1   +44.726, E3 +358194.773}
SPL {X  -165.650, Y  +433.421, Z    +0.000, E1   +45.110, E3 +358204.160}
SPL {X  -165.650, Y  +426.476, Z    +0.000, E1   +45.244, E3 +358217.664}
SPL {X  -165.650, Y  +420.418, Z    +0.000, E1   +45.128, E3 +358230.458}
SPL {X  -165.650, Y  +415.564, Z    +0.000, E1   +45.195, E3 +358240.003}
SPL {X  -165.650, Y  +410.687, Z    +0.000, E1   +44.955, E3 +358251.319}
SPL {X  -165.650, Y  +405.522, Z    +0.000, E1   +45.119, E3 +358260.879}
SPL {X  -165.650, Y  +400.300, Z    +0.000, E1   +45.439, E3 +358269.563}
SPL {X  -165.650, Y  +396.171, Z    +0.000, E1   +44.969, E3 +358280.820}
SPL {X  -165.650, Y  +390.060, Z    +0.000, E1   +45.007, E3 +358293.054}
SPL {X  -165.650, Y  +383.700, Z    +0.000, E1   +45.345, E3 +358303.978}
SPL {X  -165.650, Y  +379.225, Z    +0.000, E1   +45.073, E3 +358314.667}
SPL {X  -165.591, Y  +374.097, Z    +0.000, E1   +45.069, E3 +358325.148}
SPL {X  -165.372, Y  +368.914, Z    +0.000, E1   +45.103, E3 +358335.508}
SPL {X  -164.987, Y  +363.696, Z    +0.000, E1   +45.006, E3 +358346.731}
SPL {X  -164.256, Y  +357.053, Z    +0.000, E1   +44.969, E3 +358360.533}
SPL {X  -163.441, Y  +351.538, Z    +0.000, E1   +44.749, E3 +358372.897}
SPL {X  -162.419, Y  +345.942, Z    +0.000, E1   +44.540, E3 +358385.629}
SPL {X  -161.210, Y  +340.404, Z    +0.000, E1   +44.250, E3 +358398.454}
SPL {X  -159.961, Y  +335.460, Z    +0.000, E1   +44.205, E3 +358408.816}
SPL {X  -158.595, Y  +330.672, Z    +0.000, E1   +43.797, E3 +358420.795}
SPL {X  -157.207, Y  +326.289, Z    +0.000, E1   +43.631, E3 +358430.548}
SPL {X  -152.192, Y  +313.097, Z    +0.000, E1   +47.715, E3 +358434.101}
SPL {X  -146.385, Y  +300.967, Z    +0.000, E1   +50.402, E3 +358440.297}
SPL {X  -138.435, Y  +287.529, Z    +0.000, E1   +45.834, E3 +358502.253}
SPL {X  -134.645, Y  +282.008, Z    +0.000, E1   +45.207, E3 +358531.909}
ENDSPLINE

SPLINE
SPL {X  -154.915, Y  +319.839, Z    +0.000, E1   +31.584, E3 +358591.428}
SPL {X  -161.387, Y  +341.161, Z    +0.000, E1   +22.590, E3 +358605.274}
SPL {X  -164.566, Y  +359.576, Z    +0.000, E1   +13.425, E3 +358583.867}
SPL {X  -165.355, Y  +368.611, Z    +0.000, E1    +8.407, E3 +358587.448}
SPL {X  -165.614, Y  +375.050, Z    +0.000, E1    +4.520, E3 +358588.751}
SPL {X  -165.650, Y  +379.847, Z    +0.000, E1    +1.364, E3 +358587.101}
SPL {X  -165.650, Y  +383.246, Z    +0.000, E1    -1.216, E3 +358586.194}
SPL {X  -165.650, Y  +386.866, Z    +0.000, E1    -4.337, E3 +358586.247}
SPL {X  -165.650, Y  +392.464, Z    +0.000, E1   -10.170, E3 +358584.251}
SPL {X  -165.650, Y  +397.361, Z    +0.000, E1   -15.736, E3 +358583.582}
SPL {X  -165.650, Y  +404.553, Z    +0.000, E1   -23.488, E3 +358584.358}
SPL {X  -165.650, Y  +415.773, Z    +0.000, E1   -36.308, E3 +358580.511}
SPL {X  -165.650, Y  +456.525, Z    +0.000, E1   -55.091, E3 +358596.073}
SPL {X  -165.650, Y  +467.178, Z    +0.000, E1   -56.049, E3 +358604.810}
SPL {X  -165.650, Y  +498.574, Z    +0.000, E1   -52.082, E3 +358661.266}
ENDSPLINE

SPLINE
SPL {X  -165.650, Y  +484.983, Z    +0.000, E1   -45.406, E3 +358676.768}
ENDSPLINE

SPLINE
SPL {X  -165.650, Y  +492.090, Z    +0.000, E1   -45.292, E3 +358691.791}
SPL {X  -165.650, Y  +498.857, Z    +0.000, E1   -45.339, E3 +358705.128}
SPL {X  -165.650, Y  +504.159, Z    +0.000, E1   -45.384, E3 +358715.522}
SPL {X  -165.650, Y  +509.628, Z    +0.000, E1   -45.217, E3 +358727.706}
SPL {X  -165.650, Y  +516.157, Z    +0.000, E1   -45.240, E3 +358740.741}
SPL {X  -165.650, Y  +521.049, Z    +0.000, E1   -45.236, E3 +358750.694}
SPL {X  -165.650, Y  +527.050, Z    +0.000, E1   -45.345, E3 +358762.190}
SPL {X  -165.650, Y  +532.042, Z    +0.000, E1   -45.233, E3 +358772.933}
SPL {X  -165.650, Y  +537.290, Z    +0.000, E1   -45.204, E3 +358783.774}
SPL {X  -165.650, Y  +544.196, Z    +0.000, E1   -45.432, E3 +358796.448}
SPL {X  -165.650, Y  +548.678, Z    +0.000, E1   -45.162, E3 +358807.012}
SPL {X  -165.650, Y  +554.600, Z    +0.000, E1   -45.345, E3 +358817.989}
SPL {X  -165.650, Y  +561.799, Z    +0.000, E1   -45.312, E3 +358832.858}
SPL {X  -165.650, Y  +567.835, Z    +0.000, E1   -45.186, E3 +358845.665}
SPL {X  -165.650, Y  +573.074, Z    +0.000, E1   -45.379, E3 +358855.156}
SPL {X  -165.650, Y  +577.292, Z    +0.000, E1   -45.246, E3 +358864.419}
SPL {X  -165.650, Y  +583.131, Z    +0.000, E1   -45.255, E3 +358876.361}
SPL {X  -165.650, Y  +590.060, Z    +0.000, E1   -45.221, E3 +358890.555}
SPL {X  -165.650, Y  +596.611, Z    +0.000, E1   -45.390, E3 +358902.791}
SPL {X  -165.650, Y  +603.637, Z    +0.000, E1   -45.296, E3 +358917.710}
SPL {X  -165.650, Y  +610.850, Z    +0.000, E1   -45.208, E3 +358932.718}
SPL {X  -165.650, Y  +617.450, Z    +0.000, E1   -45.402, E3 +358944.920}
SPL {X  -165.650, Y  +622.720, Z    +0.000, E1   -45.272, E3 +358956.318}
SPL {X  -165.650, Y  +627.828, Z    +0.000, E1   -45.174, E3 +358967.275}
SPL {X  -165.650, Y  +634.620, Z    +0.000, E1   -45.438, E3 +358979.481}
SPL {X  -165.650, Y  +640.808, Z    +0.000, E1   -45.294, E3 +358992.855}
SPL {X  -165.650, Y  +646.552, Z    +0.000, E1   -45.137, E3 +359005.379}
SPL {X  -165.650, Y  +652.431, Z    +0.000, E1   -45.333, E3 +359016.134}
SPL {X  -165.650, Y  +657.443, Z    +0.000, E1   -45.316, E3 +359026.390}
SPL {X  -165.650, Y  +662.999, Z    +0.000, E1   -45.214, E3 +359038.262}
SPL {X  -165.650, Y  +668.737, Z    +0.000, E1   -45.236, E3 +359049.777}
SPL {X  -165.650, Y  +675.226, Z    +0.000, E1   -45.503, E3 +359061.280}
SPL {X  -165.597, Y  +679.672, Z    +0.000, E1   -45.206, E3 +359072.002}
SPL {X  -165.388, Y  +684.808, Z    +0.000, E1   -45.192, E3 +359082.509}
SPL {X  -165.020, Y  +689.938, Z    +0.000, E1   -45.107, E3 +359093.452}
SPL {X  -164.358, Y  +696.147, Z    +0.000, E1   -45.160, E3 +359105.718}
SPL {X  -163.631, Y  +701.286, Z    +0.000, E1   -44.994, E3 +359117.010}
SPL {X  -163.047, Y  +704.748, Z    +0.000, E1   -44.682, E3 +359125.834}
SPL {X  -161.884, Y  +710.619, Z    +0.000, E1   -44.738, E3 +359137.458}
SPL {X  -160.692, Y  +715.726, Z    +0.000, E1   -44.379, E3 +359149.781}
SPL {X  -158.938, Y  +722.175, Z    +0.000, E1   -44.121, E3 +359164.429}
SPL {X  -157.296, Y  +727.442, Z    +0.000, E1   -43.792, E3 +359176.654}
SPL {X  -153.030, Y  +738.918, Z    +0.000, E1   -47.123, E3 +359181.020}
SPL {X  -145.149, Y  +755.323, Z    +0.000, E1   -51.167, E3 +359187.152}
SPL {X  -143.038, Y  +759.047, Z    +0.000, E1   -43.157, E3 +359256.326}
SPL {X  -123.277, Y  +786.146, Z    +0.000, E1   -47.533, E3 +359312.381}
ENDSPLINE

SPLINE
SPL {X  -133.736, Y  +773.248, Z    +0.000, E1   -45.385, E3 +359377.414}
SPL {X  -160.761, Y  +715.447, Z    +0.000, E1   -23.748, E3 +359334.264}
SPL {X  -164.304, Y  +696.571, Z    +0.000, E1   -14.525, E3 +359339.488}
SPL {X  -165.498, Y  +682.585, Z    +0.000, E1    -6.769, E3 +359339.162}
SPL {X  -165.650, Y  +674.975, Z    +0.000, E1    -1.888, E3 +359337.520}
SPL {X  -165.650, Y  +671.520, Z    +0.000, E1    +0.682, E3 +359336.447}
SPL {X  -165.650, Y  +668.289, Z    +0.000, E1    +3.417, E3 +359336.289}
SPL {X  -165.650, Y  +663.040, Z    +0.000, E1    +8.602, E3 +359335.484}
SPL {X  -165.650, Y  +655.692, Z    +0.000, E1   +17.061, E3 +359334.019}
SPL {X  -165.650, Y  +646.511, Z    +0.000, E1   +26.434, E3 +359336.799}
SPL {X  -165.650, Y  +637.905, Z    +0.000, E1   +40.225, E3 +359324.924}
SPL {X  -165.650, Y  +611.479, Z    +0.000, E1   +52.226, E3 +359338.477}
SPL {X  -165.650, Y  +599.923, Z    +0.000, E1   +51.240, E3 +359355.566}
SPL {X  -165.650, Y  +553.219, Z    +0.000, E1   +52.865, E3 +359412.326}
ENDSPLINE

SPLINE
SPL {X  -165.650, Y  +569.883, Z    +0.000, E1   +45.183, E3 +359428.003}
ENDSPLINE

SPLINE
SPL {X  -165.650, Y  +561.960, Z    +0.000, E1   +45.285, E3 +359443.658}
SPL {X  -165.650, Y  +554.065, Z    +0.000, E1   +45.254, E3 +359459.720}
SPL {X  -165.650, Y  +548.074, Z    +0.000, E1   +45.245, E3 +359471.831}
SPL {X  -165.650, Y  +542.958, Z    +0.000, E1   +45.131, E3 +359482.962}
SPL {X  -165.650, Y  +535.288, Z    +0.000, E1   +45.332, E3 +359497.403}
SPL {X  -165.650, Y  +529.160, Z    +0.000, E1   +45.215, E3 +359510.383}
SPL {X  -165.650, Y  +522.672, Z    +0.000, E1   +45.331, E3 +359522.950}
SPL {X  -165.650, Y  +516.211, Z    +0.000, E1   +45.175, E3 +359536.909}
SPL {X  -165.650, Y  +509.762, Z    +0.000, E1   +45.191, E3 +359549.951}
SPL {X  -165.650, Y  +503.812, Z    +0.000, E1   +45.188, E3 +359561.990}
SPL {X  -165.650, Y  +499.646, Z    +0.000, E1   +44.886, E3 +359572.261}
ENDSPLINE

SPLINE
SPL {X  -165.650, Y  +514.834, Z    +0.000, E1   +36.829, E3 +359585.027}
ENDSPLINE

SPLINE
SPL {X  -165.650, Y  +506.421, Z    +0.000, E1   +37.886, E3 +359601.139}
SPL {X  -165.650, Y  +499.917, Z    +0.000, E1   +38.752, E3 +359612.600}
SPL {X  -165.650, Y  +493.826, Z    +0.000, E1   +39.521, E3 +359623.354}
SPL {X  -165.650, Y  +487.003, Z    +0.000, E1   +40.380, E3 +359634.808}
SPL {X  -165.650, Y  +478.382, Z    +0.000, E1   +41.628, E3 +359647.721}
SPL {X  -165.650, Y  +472.112, Z    +0.000, E1   +42.202, E3 +359658.460}
SPL {X  -165.650, Y  +466.741, Z    +0.000, E1   +42.890, E3 +359666.380}
SPL {X  -165.650, Y  +458.202, Z    +0.000, E1   +44.020, E3 +359678.168}
SPL {X  -165.650, Y  +449.099, Z    +0.000, E1   +44.871, E3 +359692.131}
SPL {X  -165.650, Y  +442.120, Z    +0.000, E1   +45.313, E3 +359703.683}
SPL {X  -165.650, Y  +436.063, Z    +0.000, E1   +44.972, E3 +359718.267}
SPL {X  -165.650, Y  +427.943, Z    +0.000, E1   +45.362, E3 +359732.304}
SPL {X  -165.650, Y  +422.523, Z    +0.000, E1   +45.103, E3 +359744.982}
SPL {X  -165.650, Y  +415.564, Z    +0.000, E1   +45.195, E3 +359758.521}
SPL {X  -165.650, Y  +410.687, Z    +0.000, E1   +44.955, E3 +359769.838}
SPL {X  -165.650, Y  +405.522, Z    +0.000, E1   +45.119, E3 +359779.398}
SPL {X  -165.650, Y  +399.216, Z    +0.000, E1   +45.246, E3 +359791.592}
SPL {X  -165.650, Y  +391.618, Z    +0.000, E1   +45.037, E3 +359808.370}
SPL {X  -165.650, Y  +383.700, Z    +0.000, E1   +45.345, E3 +359822.496}
SPL {X  -165.650, Y  +379.225, Z    +0.000, E1   +45.073, E3 +359833.185}
SPL {X  -165.591, Y  +374.097, Z    +0.000, E1   +45.069, E3 +359843.666}
SPL {X  -165.372, Y  +368.914, Z    +0.000, E1   +45.103, E3 +359854.026}
SPL {X  -164.987, Y  +363.696, Z    +0.000, E1   +45.006, E3 +359865.249}
SPL {X  -164.256, Y  +357.053, Z    +0.000, E1   +44.969, E3 +359879.052}
SPL {X  -163.441, Y  +351.538, Z    +0.000, E1   +44.749, E3 +359891.415}
SPL {X  -162.419, Y  +345.942, Z    +0.000, E1   +44.540, E3 +359904.147}
SPL {X  -161.210, Y  +340.404, Z    +0.000, E1   +44.250, E3 +359916.972}
SPL {X  -159.961, Y  +335.460, Z    +0.000, E1   +44.205, E3 +359927.335}
SPL {X  -158.595, Y  +330.672, Z    +0.000, E1   +43.797, E3 +359939.313}
SPL {X  -156.695, Y  +324.773, Z    +0.000, E1   +43.987, E3 +359950.210}
SPL {X  -148.318, Y  +304.733, Z    +0.000, E1   +49.897, E3 +359955.447}
SPL {X  -138.435, Y  +287.529, Z    +0.000, E1   +45.834, E3 +360020.771}
SPL {X  -137.083, Y  +285.505, Z    +0.000, E1   +44.955, E3 +360038.936}
ENDSPLINE

SPLINE
SPL {X  -137.518, Y  +286.149, Z    +0.000, E1   +42.648, E3 +360102.816}
SPL {X  -156.430, Y  +324.005, Z    +0.000, E1   +29.926, E3 +360107.950}
SPL {X  -161.387, Y  +341.161, Z    +0.000, E1   +22.590, E3 +360123.792}
SPL {X  -164.566, Y  +359.576, Z    +0.000, E1   +13.425, E3 +360102.385}
SPL {X  -165.355, Y  +368.611, Z    +0.000, E1    +8.407, E3 +360105.966}
SPL {X  -165.614, Y  +375.050, Z    +0.000, E1    +4.520, E3 +360107.270}
SPL {X  -165.650, Y  +379.847, Z    +0.000, E1    +1.364, E3 +360105.619}
SPL {X  -165.650, Y  +383.246, Z    +0.000, E1    -1.216, E3 +360104.713}
SPL {X  -165.650, Y  +386.866, Z    +0.000, E1    -4.337, E3 +360104.765}
SPL {X  -165.650, Y  +394.200, Z    +0.000, E1   -11.943, E3 +360102.532}
SPL {X  -165.650, Y  +405.401, Z    +0.000, E1   -24.512, E3 +360102.353}
SPL {X  -165.650, Y  +418.038, Z    +0.000, E1   -38.688, E3 +360098.580}
SPL {X  -165.650, Y  +461.620, Z    +0.000, E1   -55.594, E3 +360118.759}
SPL {X  -165.650, Y  +498.574, Z    +0.000, E1   -52.082, E3 +360179.784}
ENDSPLINE

SPLINE
SPL {X  -165.650, Y  +484.983, Z    +0.000, E1   -45.406, E3 +360195.287}
ENDSPLINE

SPLINE
SPL {X  -165.650, Y  +492.090, Z    +0.000, E1   -45.292, E3 +360210.309}
SPL {X  -165.650, Y  +498.857, Z    +0.000, E1   -45.339, E3 +360223.646}
SPL {X  -165.650, Y  +505.115, Z    +0.000, E1   -45.299, E3 +360236.595}
SPL {X  -165.650, Y  +510.931, Z    +0.000, E1   -45.250, E3 +360248.585}
SPL {X  -165.650, Y  +516.157, Z    +0.000, E1   -45.240, E3 +360259.260}
SPL {X  -165.650, Y  +521.049, Z    +0.000, E1   -45.236, E3 +360269.212}
SPL {X  -165.650, Y  +527.050, Z    +0.000, E1   -45.345, E3 +360280.709}
SPL {X  -165.650, Y  +532.042, Z    +0.000, E1   -45.233, E3 +360291.452}
SPL {X  -165.650, Y  +537.290, Z    +0.000, E1   -45.204, E3 +360302.293}
SPL {X  -165.650, Y  +544.196, Z    +0.000, E1   -45.432, E3 +360314.967}
SPL {X  -165.650, Y  +548.678, Z    +0.000, E1   -45.162, E3 +360325.531}
SPL {X  -165.650, Y  +554.600, Z    +0.000, E1   -45.345, E3 +360336.508}
SPL {X  -165.650, Y  +559.896, Z    +0.000, E1   -45.150, E3 +360348.363}
SPL {X  -165.650, Y  +566.830, Z    +0.000, E1   -45.346, E3 +360361.343}
SPL {X  -165.650, Y  +573.074, Z    +0.000, E1   -45.379, E3 +360373.674}
SPL {X  -165.650, Y  +579.360, Z    +0.000, E1   -45.300, E3 +360386.959}
SPL {X  -165.650, Y  +584.577, Z    +0.000, E1   -45.167, E3 +360398.182}
SPL {X  -165.650, Y  +590.060, Z    +0.000, E1   -45.221, E3 +360409.073}
SPL {X  -165.650, Y  +596.611, Z    +0.000, E1   -45.390, E3 +360421.310}
SPL {X  -165.650, Y  +603.637, Z    +0.000, E1   -45.296, E3 +360436.228}
SPL {X  -165.650, Y  +610.850, Z    +0.000, E1   -45.208, E3 +360451.236}
SPL {X  -165.650, Y  +617.450, Z    +0.000, E1   -45.402, E3 +360463.439}
SPL {X  -165.650, Y  +622.720, Z    +0.000, E1   -45.272, E3 +360474.837}
SPL {X  -165.650, Y  +627.828, Z    +0.000, E1   -45.174, E3 +360485.793}
SPL {X  -165.650, Y  +634.620, Z    +0.000, E1   -45.438, E3 +360497.999}
SPL {X  -165.650, Y  +640.808, Z    +0.000, E1   -45.294, E3 +360511.373}
SPL {X  -165.650, Y  +646.552, Z    +0.000, E1   -45.137, E3 +360523.898}
SPL {X  -165.650, Y  +652.431, Z    +0.000, E1   -45.333, E3 +360534.652}
SPL {X  -165.650, Y  +657.443, Z    +0.000, E1   -45.316, E3 +360544.908}
SPL {X  -165.650, Y  +662.999, Z    +0.000, E1   -45.214, E3 +360556.780}
SPL {X  -165.650, Y  +668.737, Z    +0.000, E1   -45.236, E3 +360568.295}
SPL {X  -165.650, Y  +675.226, Z    +0.000, E1   -45.503, E3 +360579.799}
SPL {X  -165.597, Y  +679.672, Z    +0.000, E1   -45.206, E3 +360590.520}
SPL {X  -165.388, Y  +684.808, Z    +0.000, E1   -45.192, E3 +360601.028}
SPL {X  -165.020, Y  +689.938, Z    +0.000, E1   -45.107, E3 +360611.970}
SPL {X  -164.358, Y  +696.147, Z    +0.000, E1   -45.160, E3 +360624.236}
SPL {X  -163.631, Y  +701.286, Z    +0.000, E1   -44.994, E3 +360635.528}
SPL {X  -162.679, Y  +706.734, Z    +0.000, E1   -44.812, E3 +360647.761}
SPL {X  -161.655, Y  +711.661, Z    +0.000, E1   -44.525, E3 +360659.142}
SPL {X  -160.692, Y  +715.726, Z    +0.000, E1   -44.379, E3 +360668.299}
SPL {X  -159.384, Y  +720.631, Z    +0.000, E1   -44.155, E3 +360679.450}
SPL {X  -158.321, Y  +724.227, Z    +0.000, E1   -43.955, E3 +360687.771}
SPL {X  -156.604, Y  +729.490, Z    +0.000, E1   -44.229, E3 +360696.937}
SPL {X  -147.100, Y  +751.668, Z    +0.000, E1   -50.624, E3 +360702.824}
SPL {X  -144.116, Y  +757.172, Z    +0.000, E1   -42.809, E3 +360772.220}
SPL {X  -127.227, Y  +781.582, Z    +0.000, E1   -46.780, E3 +360817.890}
ENDSPLINE

SPLINE
SPL {X  -133.736, Y  +773.248, Z    +0.000, E1   -45.385, E3 +360895.932}
SPL {X  -160.761, Y  +715.447, Z    +0.000, E1   -23.748, E3 +360852.782}
SPL {X  -164.304, Y  +696.571, Z    +0.000, E1   -14.525, E3 +360858.006}
SPL {X  -165.498, Y  +682.585, Z    +0.000, E1    -6.769, E3 +360857.680}
SPL {X  -165.650, Y  +674.975, Z    +0.000, E1    -1.888, E3 +360856.039}
SPL {X  -165.650, Y  +671.520, Z    +0.000, E1    +0.682, E3 +360854.966}
SPL {X  -165.650, Y  +668.289, Z    +0.000, E1    +3.417, E3 +360854.808}
SPL {X  -165.650, Y  +663.040, Z    +0.000, E1    +8.602, E3 +360854.002}
SPL {X  -165.650, Y  +655.692, Z    +0.000, E1   +17.061, E3 +360852.538}
SPL {X  -165.650, Y  +646.511, Z    +0.000, E1   +26.434, E3 +360855.318}
SPL {X  -165.650, Y  +637.905, Z    +0.000, E1   +40.225, E3 +360843.442}
SPL {X  -165.650, Y  +611.479, Z    +0.000, E1   +52.226, E3 +360856.995}
SPL {X  -165.650, Y  +599.923, Z    +0.000, E1   +51.240, E3 +360874.084}
SPL {X  -165.650, Y  +553.219, Z    +0.000, E1   +52.865, E3 +360930.845}
ENDSPLINE

SPLINE
SPL {X  -165.650, Y  +569.883, Z    +0.000, E1   +45.183, E3 +360946.521}
ENDSPLINE

SPLINE
SPL {X  -165.650, Y  +561.960, Z    +0.000, E1   +45.285, E3 +360962.177}
SPL {X  -165.650, Y  +554.065, Z    +0.000, E1   +45.254, E3 +360978.239}
SPL {X  -165.650, Y  +548.074, Z    +0.000, E1   +45.245, E3 +360990.350}
SPL {X  -165.650, Y  +542.958, Z    +0.000, E1   +45.131, E3 +361001.480}
SPL {X  -165.650, Y  +535.288, Z    +0.000, E1   +45.332, E3 +361015.921}
SPL {X  -165.650, Y  +529.160, Z    +0.000, E1   +45.215, E3 +361028.902}
SPL {X  -165.650, Y  +522.672, Z    +0.000, E1   +45.331, E3 +361041.468}
SPL {X  -165.650, Y  +516.211, Z    +0.000, E1   +45.175, E3 +361055.428}
SPL {X  -165.650, Y  +509.762, Z    +0.000, E1   +45.191, E3 +361068.470}
SPL {X  -165.650, Y  +503.812, Z    +0.000, E1   +45.188, E3 +361080.509}
SPL {X  -165.650, Y  +499.646, Z    +0.000, E1   +44.886, E3 +361090.780}
ENDSPLINE

SPLINE
SPL {X  -165.650, Y  +516.930, Z    +0.000, E1   +36.544, E3 +361099.450}
ENDSPLINE

SPLINE
SPL {X  -165.650, Y  +511.324, Z    +0.000, E1   +37.254, E3 +361110.441}
SPL {X  -165.650, Y  +504.742, Z    +0.000, E1   +38.087, E3 +361122.746}
SPL {X  -165.650, Y  +497.845, Z    +0.000, E1   +39.022, E3 +361134.821}
SPL {X  -165.650, Y  +491.819, Z    +0.000, E1   +39.756, E3 +361145.340}
SPL {X  -165.650, Y  +485.086, Z    +0.000, E1   +40.678, E3 +361156.184}
SPL {X  -165.650, Y  +476.633, Z    +0.000, E1   +41.847, E3 +361168.883}
SPL {X  -165.650, Y  +468.596, Z    +0.000, E1   +42.673, E3 +361182.146}
SPL {X  -165.650, Y  +460.562, Z    +0.000, E1   +43.733, E3 +361193.298}
SPL {X  -165.650, Y  +455.629, Z    +0.000, E1   +44.293, E3 +361200.417}
SPL {X  -165.650, Y  +449.099, Z    +0.000, E1   +44.871, E3 +361210.649}
SPL {X  -165.650, Y  +442.120, Z    +0.000, E1   +45.313, E3 +361222.201}
SPL {X  -165.650, Y  +439.103, Z    +0.000, E1   +44.726, E3 +361231.810}
SPL {X  -165.650, Y  +433.421, Z    +0.000, E1   +45.110, E3 +361241.198}
SPL {X  -165.650, Y  +426.476, Z    +0.000, E1   +45.244, E3 +361254.701}
SPL {X  -165.650, Y  +420.418, Z    +0.000, E1   +45.128, E3 +361267.495}
SPL {X  -165.650, Y  +415.564, Z    +0.000, E1   +45.195, E3 +361277.040}
SPL {X  -165.650, Y  +410.687, Z    +0.000, E1   +44.955, E3 +361288.356}
SPL {X  -165.650, Y  +402.778, Z    +0.000, E1   +45.323, E3 +361302.437}
SPL {X  -165.650, Y  +396.171, Z    +0.000, E1   +44.969, E3 +361317.857}
SPL {X  -165.650, Y  +390.060, Z    +0.000, E1   +45.007, E3 +361330.091}
SPL {X  -165.650, Y  +383.700, Z    +0.000, E1   +45.345, E3 +361341.015}
SPL {X  -165.650, Y  +379.225, Z    +0.000, E1   +45.073, E3 +361351.704}
SPL {X  -165.591, Y  +374.097, Z    +0.000, E1   +45.069, E3 +361362.185}
SPL {X  -165.372, Y  +368.914, Z    +0.000, E1   +45.103, E3 +361372.545}
SPL {X  -164.833, Y  +362.064, Z    +0.000, E1   +44.999, E3 +361387.330}
SPL {X  -164.024, Y  +355.348, Z    +0.000, E1   +45.002, E3 +361400.718}
SPL {X  -163.441, Y  +351.538, Z    +0.000, E1   +44.749, E3 +361409.934}
SPL {X  -162.419, Y  +345.942, Z    +0.000, E1   +44.540, E3 +361422.666}
SPL {X  -161.210, Y  +340.404, Z    +0.000, E1   +44.250, E3 +361435.491}
SPL {X  -159.961, Y  +335.460, Z    +0.000, E1   +44.205, E3 +361445.853}
SPL {X  -158.595, Y  +330.672, Z    +0.000, E1   +43.797, E3 +361457.832}
SPL {X  -156.695, Y  +324.773, Z    +0.000, E1   +43.987, E3 +361468.729}
SPL {X  -148.318, Y  +304.733, Z    +0.000, E1   +49.897, E3 +361473.965}
SPL {X  -138.435, Y  +287.529, Z    +0.000, E1   +45.834, E3 +361539.290}
SPL {X  -134.645, Y  +282.008, Z    +0.000, E1   +45.207, E3 +361568.946}
ENDSPLINE

SPLINE
SPL {X  -154.915, Y  +319.839, Z    +0.000, E1   +31.584, E3 +361628.465}
SPL {X  -161.387, Y  +341.161, Z    +0.000, E1   +22.590, E3 +361642.311}
SPL {X  -164.566, Y  +359.576, Z    +0.000, E1   +13.425, E3 +361620.904}
SPL {X  -165.355, Y  +368.611, Z    +0.000, E1    +8.407, E3 +361624.485}
SPL {X  -165.614, Y  +375.050, Z    +0.000, E1    +4.520, E3 +361625.789}
SPL {X  -165.650, Y  +379.847, Z    +0.000, E1    +1.364, E3 +361624.138}
SPL {X  -165.650, Y  +383.246, Z    +0.000, E1    -1.216, E3 +361623.231}
SPL {X  -165.650, Y  +386.866, Z    +0.000, E1    -4.337, E3 +361623.284}
SPL {X  -165.650, Y  +394.200, Z    +0.000, E1   -11.943, E3 +361621.051}
SPL {X  -165.650, Y  +405.401, Z    +0.000, E1   -24.512, E3 +361620.871}
SPL {X  -165.650, Y  +418.038, Z    +0.000, E1   -38.688, E3 +361617.099}
SPL {X  -165.650, Y  +461.620, Z    +0.000, E1   -55.594, E3 +361637.277}
SPL {X  -165.650, Y  +498.574, Z    +0.000, E1   -52.082, E3 +361698.303}
ENDSPLINE

SPLINE
SPL {X  -165.650, Y  +484.983, Z    +0.000, E1   -45.406, E3 +361713.805}
ENDSPLINE

SPLINE
SPL {X  -165.650, Y  +492.090, Z    +0.000, E1   -45.292, E3 +361728.828}
SPL {X  -165.650, Y  +498.857, Z    +0.000, E1   -45.339, E3 +361742.165}
SPL {X  -165.650, Y  +505.115, Z    +0.000, E1   -45.299, E3 +361755.113}
SPL {X  -165.650, Y  +510.931, Z    +0.000, E1   -45.250, E3 +361767.104}
SPL {X  -165.650, Y  +516.157, Z    +0.000, E1   -45.240, E3 +361777.778}
SPL {X  -165.650, Y  +521.049, Z    +0.000, E1   -45.236, E3 +361787.731}
SPL {X  -165.650, Y  +527.050, Z    +0.000, E1   -45.345, E3 +361799.227}
SPL {X  -165.650, Y  +532.042, Z    +0.000, E1   -45.233, E3 +361809.970}
SPL {X  -165.650, Y  +537.290, Z    +0.000, E1   -45.204, E3 +361820.811}
SPL {X  -165.650, Y  +544.196, Z    +0.000, E1   -45.432, E3 +361833.485}
SPL {X  -165.650, Y  +548.678, Z    +0.000, E1   -45.162, E3 +361844.049}
SPL {X  -165.650, Y  +554.600, Z    +0.000, E1   -45.345, E3 +361855.026}
SPL {X  -165.650, Y  +559.896, Z    +0.000, E1   -45.150, E3 +361866.882}
SPL {X  -165.650, Y  +566.830, Z    +0.000, E1   -45.346, E3 +361879.862}
SPL {X  -165.650, Y  +573.074, Z    +0.000, E1   -45.379, E3 +361892.193}
SPL {X  -165.650, Y  +579.360, Z    +0.000, E1   -45.300, E3 +361905.478}
SPL {X  -165.650, Y  +584.577, Z    +0.000, E1   -45.167, E3 +361916.701}
SPL {X  -165.650, Y  +590.060, Z    +0.000, E1   -45.221, E3 +361927.592}
SPL {X  -165.650, Y  +596.611, Z    +0.000, E1   -45.390, E3 +361939.828}
SPL {X  -165.650, Y  +603.637, Z    +0.000, E1   -45.296, E3 +361954.747}
SPL {X  -165.650, Y  +610.850, Z    +0.000, E1   -45.208, E3 +361969.755}
SPL {X  -165.650, Y  +617.450, Z    +0.000, E1   -45.402, E3 +361981.957}
SPL {X  -165.650, Y  +622.720, Z    +0.000, E1   -45.272, E3 +361993.355}
SPL {X  -165.650, Y  +627.828, Z    +0.000, E1   -45.174, E3 +362004.312}
SPL {X  -165.650, Y  +634.620, Z    +0.000, E1   -45.438, E3 +362016.518}
SPL {X  -165.650, Y  +640.808, Z    +0.000, E1   -45.294, E3 +362029.892}
SPL {X  -165.650, Y  +646.552, Z    +0.000, E1   -45.137, E3 +362042.416}
SPL {X  -165.650, Y  +652.431, Z    +0.000, E1   -45.333, E3 +362053.171}
SPL {X  -165.650, Y  +657.443, Z    +0.000, E1   -45.316, E3 +362063.427}
SPL {X  -165.650, Y  +662.999, Z    +0.000, E1   -45.214, E3 +362075.299}
SPL {X  -165.650, Y  +668.737, Z    +0.000, E1   -45.236, E3 +362086.814}
SPL {X  -165.650, Y  +675.226, Z    +0.000, E1   -45.503, E3 +362098.318}
SPL {X  -165.597, Y  +679.672, Z    +0.000, E1   -45.206, E3 +362109.039}
SPL {X  -165.388, Y  +684.808, Z    +0.000, E1   -45.192, E3 +362119.546}
SPL {X  -165.020, Y  +689.938, Z    +0.000, E1   -45.107, E3 +362130.489}
SPL {X  -164.358, Y  +696.147, Z    +0.000, E1   -45.160, E3 +362142.755}
SPL {X  -163.631, Y  +701.286, Z    +0.000, E1   -44.994, E3 +362154.047}
SPL {X  -162.679, Y  +706.734, Z    +0.000, E1   -44.812, E3 +362166.280}
SPL {X  -161.655, Y  +711.661, Z    +0.000, E1   -44.525, E3 +362177.661}
SPL {X  -160.692, Y  +715.726, Z    +0.000, E1   -44.379, E3 +362186.818}
SPL {X  -159.384, Y  +720.631, Z    +0.000, E1   -44.155, E3 +362197.968}
SPL {X  -158.321, Y  +724.227, Z    +0.000, E1   -43.955, E3 +362206.289}
SPL {X  -156.604, Y  +729.490, Z    +0.000, E1   -44.229, E3 +362215.456}
SPL {X  -147.100, Y  +751.668, Z    +0.000, E1   -50.624, E3 +362221.343}
SPL {X  -144.116, Y  +757.172, Z    +0.000, E1   -42.809, E3 +362290.739}
SPL {X  -127.227, Y  +781.582, Z    +0.000, E1   -46.780, E3 +362336.408}
ENDSPLINE

SPLINE
SPL {X  -133.736, Y  +773.248, Z    +0.000, E1   -45.385, E3 +362414.451}
SPL {X  -160.761, Y  +715.447, Z    +0.000, E1   -23.748, E3 +362371.301}
SPL {X  -164.304, Y  +696.571, Z    +0.000, E1   -14.525, E3 +362376.525}
SPL {X  -165.498, Y  +682.585, Z    +0.000, E1    -6.769, E3 +362376.199}
SPL {X  -165.650, Y  +674.975, Z    +0.000, E1    -1.888, E3 +362374.557}
SPL {X  -165.650, Y  +671.520, Z    +0.000, E1    +0.682, E3 +362373.484}
SPL {X  -165.650, Y  +668.289, Z    +0.000, E1    +3.417, E3 +362373.326}
SPL {X  -165.650, Y  +663.040, Z    +0.000, E1    +8.602, E3 +362372.521}
SPL {X  -165.650, Y  +655.692, Z    +0.000, E1   +17.061, E3 +362371.056}
SPL {X  -165.650, Y  +646.511, Z    +0.000, E1   +26.434, E3 +362373.836}
SPL {X  -165.650, Y  +637.905, Z    +0.000, E1   +40.225, E3 +362361.961}
SPL {X  -165.650, Y  +611.479, Z    +0.000, E1   +52.226, E3 +362375.514}
SPL {X  -165.650, Y  +599.923, Z    +0.000, E1   +51.240, E3 +362392.603}
SPL {X  -165.650, Y  +553.219, Z    +0.000, E1   +52.865, E3 +362449.363}
ENDSPLINE

SPLINE
SPL {X  -165.650, Y  +569.883, Z    +0.000, E1   +45.183, E3 +362465.040}
ENDSPLINE

SPLINE
SPL {X  -165.650, Y  +561.960, Z    +0.000, E1   +45.285, E3 +362480.695}
SPL {X  -165.650, Y  +554.065, Z    +0.000, E1   +45.254, E3 +362496.757}
SPL {X  -165.650, Y  +548.074, Z    +0.000, E1   +45.245, E3 +362508.868}
SPL {X  -165.650, Y  +542.958, Z    +0.000, E1   +45.131, E3 +362519.999}
SPL {X  -165.650, Y  +535.288, Z    +0.000, E1   +45.332, E3 +362534.440}
SPL {X  -165.650, Y  +529.160, Z    +0.000, E1   +45.215, E3 +362547.420}
SPL {X  -165.650, Y  +522.672, Z    +0.000, E1   +45.331, E3 +362559.987}
SPL {X  -165.650, Y  +516.211, Z    +0.000, E1   +45.175, E3 +362573.946}
SPL {X  -165.650, Y  +509.762, Z    +0.000, E1   +45.191, E3 +362586.988}
SPL {X  -165.650, Y  +503.812, Z    +0.000, E1   +45.188, E3 +362599.027}
SPL {X  -165.650, Y  +499.646, Z    +0.000, E1   +44.886, E3 +362609.298}
ENDSPLINE

SPLINE
SPL {X  -165.650, Y  +514.834, Z    +0.000, E1   +36.829, E3 +362622.064}
ENDSPLINE

SPLINE
SPL {X  -165.650, Y  +506.421, Z    +0.000, E1   +37.886, E3 +362638.176}
SPL {X  -165.650, Y  +499.917, Z    +0.000, E1   +38.752, E3 +362649.637}
SPL {X  -165.650, Y  +493.826, Z    +0.000, E1   +39.521, E3 +362660.391}
SPL {X  -165.650, Y  +487.003, Z    +0.000, E1   +40.380, E3 +362671.845}
SPL {X  -165.650, Y  +478.382, Z    +0.000, E1   +41.628, E3 +362684.758}
SPL {X  -165.650, Y  +472.112, Z    +0.000, E1   +42.202, E3 +362695.497}
SPL {X  -165.650, Y  +466.741, Z    +0.000, E1   +42.890, E3 +362703.417}
SPL {X  -165.650, Y  +458.202, Z    +0.000, E1   +44.020, E3 +362715.205}
SPL {X  -165.650, Y  +449.099, Z    +0.000, E1   +44.871, E3 +362729.168}
SPL {X  -165.650, Y  +442.120, Z    +0.000, E1   +45.313, E3 +362740.720}
SPL {X  -165.650, Y  +436.063, Z    +0.000, E1   +44.972, E3 +362755.304}
SPL {X  -165.650, Y  +427.943, Z    +0.000, E1   +45.362, E3 +362769.341}
SPL {X  -165.650, Y  +422.523, Z    +0.000, E1   +45.103, E3 +362782.020}
SPL {X  -165.650, Y  +415.564, Z    +0.000, E1   +45.195, E3 +362795.559}
SPL {X  -165.650, Y  +410.687, Z    +0.000, E1   +44.955, E3 +362806.875}
SPL {X  -165.650, Y  +405.522, Z    +0.000, E1   +45.119, E3 +362816.435}
SPL {X  -165.650, Y  +399.216, Z    +0.000, E1   +45.246, E3 +362828.629}
SPL {X  -165.650, Y  +391.618, Z    +0.000, E1   +45.037, E3 +362845.407}
SPL {X  -165.650, Y  +383.700, Z    +0.000, E1   +45.345, E3 +362859.533}
SPL {X  -165.650, Y  +379.225, Z    +0.000, E1   +45.073, E3 +362870.222}
SPL {X  -165.591, Y  +374.097, Z    +0.000, E1   +45.069, E3 +362880.703}
SPL {X  -165.372, Y  +368.914, Z    +0.000, E1   +45.103, E3 +362891.063}
SPL {X  -164.987, Y  +363.696, Z    +0.000, E1   +45.006, E3 +362902.286}
SPL {X  -164.256, Y  +357.053, Z    +0.000, E1   +44.969, E3 +362916.089}
SPL {X  -163.441, Y  +351.538, Z    +0.000, E1   +44.749, E3 +362928.452}
SPL {X  -162.419, Y  +345.942, Z    +0.000, E1   +44.540, E3 +362941.184}
SPL {X  -161.210, Y  +340.404, Z    +0.000, E1   +44.250, E3 +362954.009}
SPL {X  -159.961, Y  +335.460, Z    +0.000, E1   +44.205, E3 +362964.372}
SPL {X  -158.595, Y  +330.672, Z    +0.000, E1   +43.797, E3 +362976.350}
SPL {X  -157.207, Y  +326.289, Z    +0.000, E1   +43.631, E3 +362986.103}
SPL {X  -152.192, Y  +313.097, Z    +0.000, E1   +47.715, E3 +362989.657}
SPL {X  -146.385, Y  +300.967, Z    +0.000, E1   +50.402, E3 +362995.852}
SPL {X  -137.641, Y  +286.333, Z    +0.000, E1   +45.396, E3 +363067.344}
SPL {X  -137.518, Y  +286.149, Z    +0.000, E1   +42.648, E3 +363139.853}
ENDSPLINE

SPLINE
SPL {X  -156.430, Y  +324.005, Z    +0.000, E1   +29.926, E3 +363144.988}
SPL {X  -161.387, Y  +341.161, Z    +0.000, E1   +22.590, E3 +363160.829}
SPL {X  -164.566, Y  +359.576, Z    +0.000, E1   +13.425, E3 +363139.422}
SPL {X  -165.355, Y  +368.611, Z    +0.000, E1    +8.407, E3 +363143.003}
SPL {X  -165.614, Y  +375.050, Z    +0.000, E1    +4.520, E3 +363144.307}
SPL {X  -165.650, Y  +379.847, Z    +0.000, E1    +1.364, E3 +363142.656}
SPL {X  -165.650, Y  +384.387, Z    +0.000, E1    -2.084, E3 +363141.638}
SPL {X  -165.650, Y  +387.977, Z    +0.000, E1    -5.454, E3 +363142.123}
SPL {X  -165.650, Y  +392.464, Z    +0.000, E1   -10.170, E3 +363139.806}
SPL {X  -165.650, Y  +397.361, Z    +0.000, E1   -15.736, E3 +363139.138}
SPL {X  -165.650, Y  +404.553, Z    +0.000, E1   -23.488, E3 +363139.914}
SPL {X  -165.650, Y  +415.773, Z    +0.000, E1   -36.308, E3 +363136.066}
SPL {X  -165.650, Y  +461.620, Z    +0.000, E1   -55.594, E3 +363155.796}
SPL {X  -165.650, Y  +498.574, Z    +0.000, E1   -52.082, E3 +363216.821}
ENDSPLINE

SPLINE
SPL {X  -165.650, Y  +484.983, Z    +0.000, E1   -45.406, E3 +363232.324}
ENDSPLINE

SPLINE
SPL {X  -165.650, Y  +492.090, Z    +0.000, E1   -45.292, E3 +363247.346}
SPL {X  -165.650, Y  +498.857, Z    +0.000, E1   -45.339, E3 +363260.683}
SPL {X  -165.650, Y  +505.115, Z    +0.000, E1   -45.299, E3 +363273.632}
SPL {X  -165.650, Y  +510.931, Z    +0.000, E1   -45.250, E3 +363285.622}
SPL {X  -165.650, Y  +516.157, Z    +0.000, E1   -45.240, E3 +363296.297}
SPL {X  -165.650, Y  +521.049, Z    +0.000, E1   -45.236, E3 +363306.249}
SPL {X  -165.650, Y  +527.050, Z    +0.000, E1   -45.345, E3 +363317.746}
SPL {X  -165.650, Y  +532.042, Z    +0.000, E1   -45.233, E3 +363328.489}
SPL {X  -165.650, Y  +537.290, Z    +0.000, E1   -45.204, E3 +363339.330}
SPL {X  -165.650, Y  +544.196, Z    +0.000, E1   -45.432, E3 +363352.004}
SPL {X  -165.650, Y  +548.678, Z    +0.000, E1   -45.162, E3 +363362.568}
SPL {X  -165.650, Y  +554.600, Z    +0.000, E1   -45.345, E3 +363373.545}
SPL {X  -165.650, Y  +559.896, Z    +0.000, E1   -45.150, E3 +363385.400}
SPL {X  -165.650, Y  +566.830, Z    +0.000, E1   -45.346, E3 +363398.380}
SPL {X  -165.650, Y  +573.074, Z    +0.000, E1   -45.379, E3 +363410.711}
SPL {X  -165.650, Y  +579.360, Z    +0.000, E1   -45.300, E3 +363423.996}
SPL {X  -165.650, Y  +584.577, Z    +0.000, E1   -45.167, E3 +363435.219}
SPL {X  -165.650, Y  +590.060, Z    +0.000, E1   -45.221, E3 +363446.110}
SPL {X  -165.650, Y  +596.611, Z    +0.000, E1   -45.390, E3 +363458.347}
SPL {X  -165.650, Y  +603.637, Z    +0.000, E1   -45.296, E3 +363473.265}
SPL {X  -165.650, Y  +610.850, Z    +0.000, E1   -45.208, E3 +363488.273}
SPL {X  -165.650, Y  +617.450, Z    +0.000, E1   -45.402, E3 +363500.476}
SPL {X  -165.650, Y  +622.720, Z    +0.000, E1   -45.272, E3 +363511.874}
SPL {X  -165.650, Y  +627.828, Z    +0.000, E1   -45.174, E3 +363522.830}
SPL {X  -165.650, Y  +634.620, Z    +0.000, E1   -45.438, E3 +363535.036}
SPL {X  -165.650, Y  +640.808, Z    +0.000, E1   -45.294, E3 +363548.410}
SPL {X  -165.650, Y  +646.552, Z    +0.000, E1   -45.137, E3 +363560.935}
SPL {X  -165.650, Y  +652.431, Z    +0.000, E1   -45.333, E3 +363571.689}
SPL {X  -165.650, Y  +657.443, Z    +0.000, E1   -45.316, E3 +363581.945}
SPL {X  -165.650, Y  +662.999, Z    +0.000, E1   -45.214, E3 +363593.817}
SPL {X  -165.650, Y  +668.737, Z    +0.000, E1   -45.236, E3 +363605.332}
SPL {X  -165.650, Y  +675.226, Z    +0.000, E1   -45.503, E3 +363616.836}
SPL {X  -165.597, Y  +679.672, Z    +0.000, E1   -45.206, E3 +363627.557}
SPL {X  -165.388, Y  +684.808, Z    +0.000, E1   -45.192, E3 +363638.065}
SPL {X  -165.020, Y  +689.938, Z    +0.000, E1   -45.107, E3 +363649.008}
SPL {X  -164.358, Y  +696.147, Z    +0.000, E1   -45.160, E3 +363661.273}
SPL {X  -163.631, Y  +701.286, Z    +0.000, E1   -44.994, E3 +363672.565}
SPL {X  -162.679, Y  +706.734, Z    +0.000, E1   -44.812, E3 +363684.798}
SPL {X  -161.655, Y  +711.661, Z    +0.000, E1   -44.525, E3 +363696.179}
SPL {X  -160.692, Y  +715.726, Z    +0.000, E1   -44.379, E3 +363705.336}
SPL {X  -159.384, Y  +720.631, Z    +0.000, E1   -44.155, E3 +363716.487}
SPL {X  -158.321, Y  +724.227, Z    +0.000, E1   -43.955, E3 +363724.808}
SPL {X  -156.604, Y  +729.490, Z    +0.000, E1   -44.229, E3 +363733.974}
SPL {X  -147.100, Y  +751.668, Z    +0.000, E1   -50.624, E3 +363739.861}
SPL {X  -144.116, Y  +757.172, Z    +0.000, E1   -42.809, E3 +363809.257}
SPL {X  -127.227, Y  +781.582, Z    +0.000, E1   -46.780, E3 +363854.927}
ENDSPLINE

SPLINE
SPL {X  -133.736, Y  +773.248, Z    +0.000, E1   -45.385, E3 +363932.969}
SPL {X  -160.761, Y  +715.447, Z    +0.000, E1   -23.748, E3 +363889.819}
SPL {X  -164.304, Y  +696.571, Z    +0.000, E1   -14.525, E3 +363895.043}
SPL {X  -165.498, Y  +682.585, Z    +0.000, E1    -6.769, E3 +363894.717}
SPL {X  -165.650, Y  +674.975, Z    +0.000, E1    -1.888, E3 +363893.076}
SPL {X  -165.650, Y  +671.520, Z    +0.000, E1    +0.682, E3 +363892.003}
SPL {X  -165.650, Y  +668.289, Z    +0.000, E1    +3.417, E3 +363891.845}
SPL {X  -165.650, Y  +663.040, Z    +0.000, E1    +8.602, E3 +363891.040}
SPL {X  -165.650, Y  +655.692, Z    +0.000, E1   +17.061, E3 +363889.575}
SPL {X  -165.650, Y  +646.511, Z    +0.000, E1   +26.434, E3 +363892.355}
SPL {X  -165.650, Y  +637.905, Z    +0.000, E1   +40.225, E3 +363880.480}
SPL {X  -165.650, Y  +611.479, Z    +0.000, E1   +52.226, E3 +363894.032}
SPL {X  -165.650, Y  +599.923, Z    +0.000, E1   +51.240, E3 +363911.121}
SPL {X  -165.650, Y  +553.219, Z    +0.000, E1   +52.865, E3 +363967.882}
ENDSPLINE

SPLINE
SPL {X  -165.650, Y  +569.883, Z    +0.000, E1   +45.183, E3 +363983.558}
ENDSPLINE

SPLINE
SPL {X  -165.650, Y  +561.960, Z    +0.000, E1   +45.285, E3 +363999.214}
SPL {X  -165.650, Y  +554.065, Z    +0.000, E1   +45.254, E3 +364015.276}
SPL {X  -165.650, Y  +548.074, Z    +0.000, E1   +45.245, E3 +364027.387}
SPL {X  -165.650, Y  +542.958, Z    +0.000, E1   +45.131, E3 +364038.517}
SPL {X  -165.650, Y  +535.288, Z    +0.000, E1   +45.332, E3 +364052.958}
SPL {X  -165.650, Y  +529.160, Z    +0.000, E1   +45.215, E3 +364065.939}
SPL {X  -165.650, Y  +522.672, Z    +0.000, E1   +45.331, E3 +364078.505}
SPL {X  -165.650, Y  +516.211, Z    +0.000, E1   +45.175, E3 +364092.465}
SPL {X  -165.650, Y  +509.762, Z    +0.000, E1   +45.191, E3 +364105.507}
SPL {X  -165.650, Y  +503.812, Z    +0.000, E1   +45.188, E3 +364117.546}
SPL {X  -165.650, Y  +499.646, Z    +0.000, E1   +44.886, E3 +364127.817}
ENDSPLINE

SPLINE
SPL {X  -165.650, Y  +516.930, Z    +0.000, E1   +36.544, E3 +364136.487}
ENDSPLINE

SPLINE
SPL {X  -165.650, Y  +511.324, Z    +0.000, E1   +37.254, E3 +364147.478}
SPL {X  -165.650, Y  +504.742, Z    +0.000, E1   +38.087, E3 +364159.783}
SPL {X  -165.650, Y  +497.845, Z    +0.000, E1   +39.022, E3 +364171.858}
SPL {X  -165.650, Y  +491.819, Z    +0.000, E1   +39.756, E3 +364182.377}
SPL {X  -165.650, Y  +485.086, Z    +0.000, E1   +40.678, E3 +364193.221}
SPL {X  -165.650, Y  +476.633, Z    +0.000, E1   +41.847, E3 +364205.920}
SPL {X  -165.650, Y  +468.596, Z    +0.000, E1   +42.673, E3 +364219.183}
SPL {X  -165.650, Y  +460.562, Z    +0.000, E1   +43.733, E3 +364230.335}
SPL {X  -165.650, Y  +455.629, Z    +0.000, E1   +44.293, E3 +364237.454}
SPL {X  -165.650, Y  +449.099, Z    +0.000, E1   +44.871, E3 +364247.686}
SPL {X  -165.650, Y  +442.120, Z    +0.000, E1   +45.313, E3 +364259.238}
SPL {X  -165.650, Y  +439.103, Z    +0.000, E1   +44.726, E3 +364268.847}
SPL {X  -165.650, Y  +433.421, Z    +0.000, E1   +45.110, E3 +364278.235}
SPL {X  -165.650, Y  +426.476, Z    +0.000, E1   +45.244, E3 +364291.738}
SPL {X  -165.650, Y  +420.418, Z    +0.000, E1   +45.128, E3 +364304.532}
SPL {X  -165.650, Y  +415.564, Z    +0.000, E1   +45.195, E3 +364314.077}
SPL {X  -165.650, Y  +410.687, Z    +0.000, E1   +44.955, E3 +364325.393}
SPL {X  -165.650, Y  +402.778, Z    +0.000, E1   +45.323, E3 +364339.474}
SPL {X  -165.650, Y  +396.171, Z    +0.000, E1   +44.969, E3 +364354.894}
SPL {X  -165.650, Y  +390.060, Z    +0.000, E1   +45.007, E3 +364367.128}
SPL {X  -165.650, Y  +383.700, Z    +0.000, E1   +45.345, E3 +364378.052}
SPL {X  -165.650, Y  +379.225, Z    +0.000, E1   +45.073, E3 +364388.741}
SPL {X  -165.591, Y  +374.097, Z    +0.000, E1   +45.069, E3 +364399.222}
SPL {X  -165.372, Y  +368.914, Z    +0.000, E1   +45.103, E3 +364409.582}
SPL {X  -164.833, Y  +362.064, Z    +0.000, E1   +44.999, E3 +364424.367}
SPL {X  -164.024, Y  +355.348, Z    +0.000, E1   +45.002, E3 +364437.755}
SPL {X  -163.441, Y  +351.538, Z    +0.000, E1   +44.749, E3 +364446.971}
SPL {X  -162.419, Y  +345.942, Z    +0.000, E1   +44.540, E3 +364459.703}
SPL {X  -161.210, Y  +340.404, Z    +0.000, E1   +44.250, E3 +364472.528}
SPL {X  -159.961, Y  +335.460, Z    +0.000, E1   +44.205, E3 +364482.890}
SPL {X  -158.595, Y  +330.672, Z    +0.000, E1   +43.797, E3 +364494.869}
SPL {X  -157.207, Y  +326.289, Z    +0.000, E1   +43.631, E3 +364504.622}
SPL {X  -152.192, Y  +313.097, Z    +0.000, E1   +47.715, E3 +364508.175}
SPL {X  -146.385, Y  +300.967, Z    +0.000, E1   +50.402, E3 +364514.371}
SPL {X  -137.641, Y  +286.333, Z    +0.000, E1   +45.396, E3 +364585.862}
SPL {X  -137.518, Y  +286.149, Z    +0.000, E1   +42.648, E3 +364658.371}
ENDSPLINE

SPLINE
SPL {X  -156.430, Y  +324.005, Z    +0.000, E1   +29.926, E3 +364663.506}
SPL {X  -161.387, Y  +341.161, Z    +0.000, E1   +22.590, E3 +364679.348}
SPL {X  -164.566, Y  +359.576, Z    +0.000, E1   +13.425, E3 +364657.941}
SPL {X  -165.355, Y  +368.611, Z    +0.000, E1    +8.407, E3 +364661.522}
SPL {X  -165.614, Y  +375.050, Z    +0.000, E1    +4.520, E3 +364662.826}
SPL {X  -165.650, Y  +379.847, Z    +0.000, E1    +1.364, E3 +364661.175}
SPL {X  -165.650, Y  +383.246, Z    +0.000, E1    -1.216, E3 +364660.269}
SPL {X  -165.650, Y  +386.866, Z    +0.000, E1    -4.337, E3 +364660.321}
SPL {X  -165.650, Y  +392.464, Z    +0.000, E1   -10.170, E3 +364658.325}
SPL {X  -165.650, Y  +397.361, Z    +0.000, E1   -15.736, E3 +364657.656}
SPL {X  -165.650, Y  +404.553, Z    +0.000, E1   -23.488, E3 +364658.432}
SPL {X  -165.650, Y  +415.773, Z    +0.000, E1   -36.308, E3 +364654.585}
SPL {X  -165.650, Y  +461.620, Z    +0.000, E1   -55.594, E3 +364674.314}
SPL {X  -165.650, Y  +498.574, Z    +0.000, E1   -52.082, E3 +364735.340}
ENDSPLINE

SPLINE
SPL {X  -165.650, Y  +484.983, Z    +0.000, E1   -45.406, E3 +364750.842}
ENDSPLINE

SPLINE
SPL {X  -165.650, Y  +492.090, Z    +0.000, E1   -45.292, E3 +364765.865}
SPL {X  -165.650, Y  +498.857, Z    +0.000, E1   -45.339, E3 +364779.202}
SPL {X  -165.650, Y  +505.115, Z    +0.000, E1   -45.299, E3 +364792.150}
SPL {X  -165.650, Y  +510.931, Z    +0.000, E1   -45.250, E3 +364804.141}
SPL {X  -165.650, Y  +516.157, Z    +0.000, E1   -45.240, E3 +364814.815}
SPL {X  -165.650, Y  +521.049, Z    +0.000, E1   -45.236, E3 +364824.768}
SPL {X  -165.650, Y  +527.050, Z    +0.000, E1   -45.345, E3 +364836.264}
SPL {X  -165.650, Y  +532.042, Z    +0.000, E1   -45.233, E3 +364847.007}
SPL {X  -165.650, Y  +537.290, Z    +0.000, E1   -45.204, E3 +364857.848}
SPL {X  -165.650, Y  +544.196, Z    +0.000, E1   -45.432, E3 +364870.522}
SPL {X  -165.650, Y  +548.678, Z    +0.000, E1   -45.162, E3 +364881.086}
SPL {X  -165.650, Y  +554.600, Z    +0.000, E1   -45.345, E3 +364892.063}
SPL {X  -165.650, Y  +559.896, Z    +0.000, E1   -45.150, E3 +364903.919}
SPL {X  -165.650, Y  +566.830, Z    +0.000, E1   -45.346, E3 +364916.899}
SPL {X  -165.650, Y  +573.074, Z    +0.000, E1   -45.379, E3 +364929.230}
SPL {X  -165.650, Y  +579.360, Z    +0.000, E1   -45.300, E3 +364942.515}
SPL {X  -165.650, Y  +584.577, Z    +0.000, E1   -45.167, E3 +364953.738}
SPL {X  -165.650, Y  +590.060, Z    +0.000, E1   -45.221, E3 +364964.629}
SPL {X  -165.650, Y  +596.611, Z    +0.000, E1   -45.390, E3 +364976.865}
SPL {X  -165.650, Y  +603.637, Z    +0.000, E1   -45.296, E3 +364991.784}
SPL {X  -165.650, Y  +610.850, Z    +0.000, E1   -45.208, E3 +365006.792}
SPL {X  -165.650, Y  +617.450, Z    +0.000, E1   -45.402, E3 +365018.994}
SPL {X  -165.650, Y  +622.720, Z    +0.000, E1   -45.272, E3 +365030.392}
SPL {X  -165.650, Y  +627.828, Z    +0.000, E1   -45.174, E3 +365041.349}
SPL {X  -165.650, Y  +634.620, Z    +0.000, E1   -45.438, E3 +365053.555}
SPL {X  -165.650, Y  +640.808, Z    +0.000, E1   -45.294, E3 +365066.929}
SPL {X  -165.650, Y  +646.552, Z    +0.000, E1   -45.137, E3 +365079.453}
SPL {X  -165.650, Y  +652.431, Z    +0.000, E1   -45.333, E3 +365090.208}
SPL {X  -165.650, Y  +657.443, Z    +0.000, E1   -45.316, E3 +365100.464}
SPL {X  -165.650, Y  +662.999, Z    +0.000, E1   -45.214, E3 +365112.336}
SPL {X  -165.650, Y  +668.737, Z    +0.000, E1   -45.236, E3 +365123.851}
SPL {X  -165.650, Y  +675.226, Z    +0.000, E1   -45.503, E3 +365135.355}
SPL {X  -165.597, Y  +679.672, Z    +0.000, E1   -45.206, E3 +365146.076}
SPL {X  -165.388, Y  +684.808, Z    +0.000, E1   -45.192, E3 +365156.583}
SPL {X  -165.020, Y  +689.938, Z    +0.000, E1   -45.107, E3 +365167.526}
SPL {X  -164.358, Y  +696.147, Z    +0.000, E1   -45.160, E3 +365179.792}
SPL {X  -163.631, Y  +701.286, Z    +0.000, E1   -44.994, E3 +365191.084}
SPL {X  -162.679, Y  +706.734, Z    +0.000, E1   -44.812, E3 +365203.317}
SPL {X  -161.655, Y  +711.661, Z    +0.000, E1   -44.525, E3 +365214.698}
SPL {X  -160.692, Y  +715.726, Z    +0.000, E1   -44.379, E3 +365223.855}
SPL {X  -159.384, Y  +720.631, Z    +0.000, E1   -44.155, E3 +365235.005}
SPL {X  -158.321, Y  +724.227, Z    +0.000, E1   -43.955, E3 +365243.326}
SPL {X  -156.604, Y  +729.490, Z    +0.000, E1   -44.229, E3 +365252.493}
SPL {X  -147.100, Y  +751.668, Z    +0.000, E1   -50.624, E3 +365258.380}
SPL {X  -144.116, Y  +757.172, Z    +0.000, E1   -42.809, E3 +365327.776}
SPL {X  -127.227, Y  +781.582, Z    +0.000, E1   -46.780, E3 +365373.445}
ENDSPLINE

SPLINE
SPL {X  -133.736, Y  +773.248, Z    +0.000, E1   -45.385, E3 +365451.488}
SPL {X  -160.761, Y  +715.447, Z    +0.000, E1   -23.748, E3 +365408.338}
SPL {X  -164.304, Y  +696.571, Z    +0.000, E1   -14.525, E3 +365413.562}
SPL {X  -165.498, Y  +682.585, Z    +0.000, E1    -6.769, E3 +365413.236}
SPL {X  -165.650, Y  +674.975, Z    +0.000, E1    -1.888, E3 +365411.594}
SPL {X  -165.650, Y  +671.520, Z    +0.000, E1    +0.682, E3 +365410.522}
SPL {X  -165.650, Y  +668.289, Z    +0.000, E1    +3.417, E3 +365410.363}
SPL {X  -165.650, Y  +663.040, Z    +0.000, E1    +8.602, E3 +365409.558}
SPL {X  -165.650, Y  +655.692, Z    +0.000, E1   +17.061, E3 +365408.093}
SPL {X  -165.650, Y  +646.511, Z    +0.000, E1   +26.434, E3 +365410.873}
SPL {X  -165.650, Y  +637.905, Z    +0.000, E1   +40.225, E3 +365398.998}
SPL {X  -165.650, Y  +611.479, Z    +0.000, E1   +52.226, E3 +365412.551}
SPL {X  -165.650, Y  +599.923, Z    +0.000, E1   +51.240, E3 +365429.640}
SPL {X  -165.650, Y  +553.219, Z    +0.000, E1   +52.865, E3 +365486.400}
ENDSPLINE

SPLINE
SPL {X  -165.650, Y  +569.883, Z    +0.000, E1   +45.183, E3 +365502.077}
ENDSPLINE

SPLINE
SPL {X  -165.650, Y  +561.960, Z    +0.000, E1   +45.285, E3 +365517.732}
SPL {X  -165.650, Y  +554.065, Z    +0.000, E1   +45.254, E3 +365533.794}
SPL {X  -165.650, Y  +548.074, Z    +0.000, E1   +45.245, E3 +365545.905}
SPL {X  -165.650, Y  +542.958, Z    +0.000, E1   +45.131, E3 +365557.036}
SPL {X  -165.650, Y  +535.288, Z    +0.000, E1   +45.332, E3 +365571.477}
SPL {X  -165.650, Y  +529.160, Z    +0.000, E1   +45.215, E3 +365584.458}
SPL {X  -165.650, Y  +522.672, Z    +0.000, E1   +45.331, E3 +365597.024}
SPL {X  -165.650, Y  +516.211, Z    +0.000, E1   +45.175, E3 +365610.983}
SPL {X  -165.650, Y  +509.762, Z    +0.000, E1   +45.191, E3 +365624.025}
SPL {X  -165.650, Y  +503.812, Z    +0.000, E1   +45.188, E3 +365636.064}
SPL {X  -165.650, Y  +499.646, Z    +0.000, E1   +44.886, E3 +365646.335}
ENDSPLINE

SPLINE
SPL {X  -165.650, Y  +516.930, Z    +0.000, E1   +36.544, E3 +365655.006}
ENDSPLINE

SPLINE
SPL {X  -165.650, Y  +511.324, Z    +0.000, E1   +37.254, E3 +365665.997}
SPL {X  -165.650, Y  +504.742, Z    +0.000, E1   +38.087, E3 +365678.302}
SPL {X  -165.650, Y  +497.845, Z    +0.000, E1   +39.022, E3 +365690.377}
SPL {X  -165.650, Y  +491.819, Z    +0.000, E1   +39.756, E3 +365700.896}
SPL {X  -165.650, Y  +485.086, Z    +0.000, E1   +40.678, E3 +365711.740}
SPL {X  -165.650, Y  +476.633, Z    +0.000, E1   +41.847, E3 +365724.439}
SPL {X  -165.650, Y  +468.596, Z    +0.000, E1   +42.673, E3 +365737.701}
SPL {X  -165.650, Y  +460.562, Z    +0.000, E1   +43.733, E3 +365748.854}
SPL {X  -165.650, Y  +455.629, Z    +0.000, E1   +44.293, E3 +365755.973}
SPL {X  -165.650, Y  +449.099, Z    +0.000, E1   +44.871, E3 +365766.205}
SPL {X  -165.650, Y  +442.120, Z    +0.000, E1   +45.313, E3 +365777.757}
SPL {X  -165.650, Y  +439.103, Z    +0.000, E1   +44.726, E3 +365787.365}
SPL {X  -165.650, Y  +433.421, Z    +0.000, E1   +45.110, E3 +365796.753}
SPL {X  -165.650, Y  +426.476, Z    +0.000, E1   +45.244, E3 +365810.257}
SPL {X  -165.650, Y  +420.418, Z    +0.000, E1   +45.128, E3 +365823.050}
SPL {X  -165.650, Y  +415.564, Z    +0.000, E1   +45.195, E3 +365832.596}
SPL {X  -165.650, Y  +410.687, Z    +0.000, E1   +44.955, E3 +365843.912}
SPL {X  -165.650, Y  +402.778, Z    +0.000, E1   +45.323, E3 +365857.992}
SPL {X  -165.650, Y  +396.171, Z    +0.000, E1   +44.969, E3 +365873.413}
SPL {X  -165.650, Y  +390.060, Z    +0.000, E1   +45.007, E3 +365885.647}
SPL {X  -165.650, Y  +383.700, Z    +0.000, E1   +45.345, E3 +365896.570}
SPL {X  -165.650, Y  +379.225, Z    +0.000, E1   +45.073, E3 +365907.259}
SPL {X  -165.591, Y  +374.097, Z    +0.000, E1   +45.069, E3 +365917.740}
SPL {X  -165.372, Y  +368.914, Z    +0.000, E1   +45.103, E3 +365928.100}
SPL {X  -164.833, Y  +362.064, Z    +0.000, E1   +44.999, E3 +365942.885}
SPL {X  -164.024, Y  +355.348, Z    +0.000, E1   +45.002, E3 +365956.274}
SPL {X  -163.441, Y  +351.538, Z    +0.000, E1   +44.749, E3 +365965.490}
SPL {X  -162.419, Y  +345.942, Z    +0.000, E1   +44.540, E3 +365978.221}
SPL {X  -161.210, Y  +340.404, Z    +0.000, E1   +44.250, E3 +365991.046}
SPL {X  -159.961, Y  +335.460, Z    +0.000, E1   +44.205, E3 +366001.409}
SPL {X  -158.595, Y  +330.672, Z    +0.000, E1   +43.797, E3 +366013.387}
SPL {X  -156.695, Y  +324.773, Z    +0.000, E1   +43.987, E3 +366024.284}
SPL {X  -148.318, Y  +304.733, Z    +0.000, E1   +49.897, E3 +366029.521}
SPL {X  -138.435, Y  +287.529, Z    +0.000, E1   +45.834, E3 +366094.845}
SPL {X  -134.645, Y  +282.008, Z    +0.000, E1   +45.207, E3 +366124.501}
ENDSPLINE

SPLINE
SPL {X  -154.915, Y  +319.839, Z    +0.000, E1   +31.584, E3 +366184.021}
SPL {X  -161.387, Y  +341.161, Z    +0.000, E1   +22.590, E3 +366197.866}
SPL {X  -164.566, Y  +359.576, Z    +0.000, E1   +13.425, E3 +366176.459}
SPL {X  -165.355, Y  +368.611, Z    +0.000, E1    +8.407, E3 +366180.040}
SPL {X  -165.614, Y  +375.050, Z    +0.000, E1    +4.520, E3 +366181.344}
SPL {X  -165.650, Y  +379.847, Z    +0.000, E1    +1.364, E3 +366179.693}
SPL {X  -165.650, Y  +383.246, Z    +0.000, E1    -1.216, E3 +366178.787}
SPL {X  -165.650, Y  +386.866, Z    +0.000, E1    -4.337, E3 +366178.839}
SPL {X  -165.650, Y  +394.200, Z    +0.000, E1   -11.943, E3 +366176.606}
SPL {X  -165.650, Y  +405.401, Z    +0.000, E1   -24.512, E3 +366176.427}
SPL {X  -165.650, Y  +418.038, Z    +0.000, E1   -38.688, E3 +366172.654}
SPL {X  -165.650, Y  +461.620, Z    +0.000, E1   -55.594, E3 +366192.833}
SPL {X  -165.650, Y  +498.574, Z    +0.000, E1   -52.082, E3 +366253.858}
ENDSPLINE

SPLINE
SPL {X  -165.650, Y  +484.983, Z    +0.000, E1   -45.406, E3 +366269.361}
ENDSPLINE

SPLINE
SPL {X  -165.650, Y  +492.090, Z    +0.000, E1   -45.292, E3 +366284.383}
SPL {X  -165.650, Y  +498.857, Z    +0.000, E1   -45.339, E3 +366297.720}
SPL {X  -165.650, Y  +505.115, Z    +0.000, E1   -45.299, E3 +366310.669}
SPL {X  -165.650, Y  +510.931, Z    +0.000, E1   -45.250, E3 +366322.659}
SPL {X  -165.650, Y  +516.157, Z    +0.000, E1   -45.240, E3 +366333.334}
SPL {X  -165.650, Y  +521.049, Z    +0.000, E1   -45.236, E3 +366343.286}
SPL {X  -165.650, Y  +527.050, Z    +0.000, E1   -45.345, E3 +366354.783}
SPL {X  -165.650, Y  +532.042, Z    +0.000, E1   -45.233, E3 +366365.526}
SPL {X  -165.650, Y  +537.290, Z    +0.000, E1   -45.204, E3 +366376.367}
SPL {X  -165.650, Y  +544.196, Z    +0.000, E1   -45.432, E3 +366389.041}
SPL {X  -165.650, Y  +548.678, Z    +0.000, E1   -45.162, E3 +366399.605}
SPL {X  -165.650, Y  +554.600, Z    +0.000, E1   -45.345, E3 +366410.582}
SPL {X  -165.650, Y  +561.799, Z    +0.000, E1   -45.312, E3 +366425.451}
SPL {X  -165.650, Y  +567.835, Z    +0.000, E1   -45.186, E3 +366438.257}
SPL {X  -165.650, Y  +573.074, Z    +0.000, E1   -45.379, E3 +366447.748}
SPL {X  -165.650, Y  +577.292, Z    +0.000, E1   -45.246, E3 +366457.012}
SPL {X  -165.650, Y  +583.131, Z    +0.000, E1   -45.255, E3 +366468.954}
SPL {X  -165.650, Y  +590.060, Z    +0.000, E1   -45.221, E3 +366483.147}
SPL {X  -165.650, Y  +596.611, Z    +0.000, E1   -45.390, E3 +366495.384}
SPL {X  -165.650, Y  +603.637, Z    +0.000, E1   -45.296, E3 +366510.302}
SPL {X  -165.650, Y  +610.850, Z    +0.000, E1   -45.208, E3 +366525.311}
SPL {X  -165.650, Y  +617.450, Z    +0.000, E1   -45.402, E3 +366537.513}
SPL {X  -165.650, Y  +622.720, Z    +0.000, E1   -45.272, E3 +366548.911}
SPL {X  -165.650, Y  +627.828, Z    +0.000, E1   -45.174, E3 +366559.867}
SPL {X  -165.650, Y  +634.620, Z    +0.000, E1   -45.438, E3 +366572.073}
SPL {X  -165.650, Y  +640.808, Z    +0.000, E1   -45.294, E3 +366585.447}
SPL {X  -165.650, Y  +646.552, Z    +0.000, E1   -45.137, E3 +366597.972}
SPL {X  -165.650, Y  +652.431, Z    +0.000, E1   -45.333, E3 +366608.726}
SPL {X  -165.650, Y  +657.443, Z    +0.000, E1   -45.316, E3 +366618.983}
SPL {X  -165.650, Y  +662.999, Z    +0.000, E1   -45.214, E3 +366630.855}
SPL {X  -165.650, Y  +668.737, Z    +0.000, E1   -45.236, E3 +366642.369}
SPL {X  -165.650, Y  +675.226, Z    +0.000, E1   -45.503, E3 +366653.873}
SPL {X  -165.597, Y  +679.672, Z    +0.000, E1   -45.206, E3 +366664.594}
SPL {X  -165.388, Y  +684.808, Z    +0.000, E1   -45.192, E3 +366675.102}
SPL {X  -165.020, Y  +689.938, Z    +0.000, E1   -45.107, E3 +366686.045}
SPL {X  -164.358, Y  +696.147, Z    +0.000, E1   -45.160, E3 +366698.310}
SPL {X  -163.631, Y  +701.286, Z    +0.000, E1   -44.994, E3 +366709.602}
SPL {X  -163.047, Y  +704.748, Z    +0.000, E1   -44.682, E3 +366718.426}
SPL {X  -161.884, Y  +710.619, Z    +0.000, E1   -44.738, E3 +366730.051}
SPL {X  -160.692, Y  +715.726, Z    +0.000, E1   -44.379, E3 +366742.374}
SPL {X  -159.384, Y  +720.631, Z    +0.000, E1   -44.155, E3 +366753.524}
SPL {X  -157.745, Y  +726.062, Z    +0.000, E1   -43.902, E3 +366766.010}
SPL {X  -153.030, Y  +738.918, Z    +0.000, E1   -47.123, E3 +366773.612}
SPL {X  -145.149, Y  +755.323, Z    +0.000, E1   -51.167, E3 +366779.744}
SPL {X  -143.038, Y  +759.047, Z    +0.000, E1   -43.157, E3 +366848.918}
SPL {X  -123.277, Y  +786.146, Z    +0.000, E1   -47.533, E3 +366904.974}
ENDSPLINE

SPLINE
SPL {X  -133.736, Y  +773.248, Z    +0.000, E1   -45.385, E3 +366970.006}
SPL {X  -160.761, Y  +715.447, Z    +0.000, E1   -23.748, E3 +366926.856}
SPL {X  -164.304, Y  +696.571, Z    +0.000, E1   -14.525, E3 +366932.080}
SPL {X  -165.498, Y  +682.585, Z    +0.000, E1    -6.769, E3 +366931.755}
SPL {X  -165.650, Y  +674.975, Z    +0.000, E1    -1.888, E3 +366930.113}
SPL {X  -165.650, Y  +671.520, Z    +0.000, E1    +0.682, E3 +366929.040}
SPL {X  -165.650, Y  +668.289, Z    +0.000, E1    +3.417, E3 +366928.882}
SPL {X  -165.650, Y  +663.040, Z    +0.000, E1    +8.602, E3 +366928.077}
SPL {X  -165.650, Y  +655.692, Z    +0.000, E1   +17.061, E3 +366926.612}
SPL {X  -165.650, Y  +646.511, Z    +0.000, E1   +26.434, E3 +366929.392}
SPL {X  -165.650, Y  +637.905, Z    +0.000, E1   +40.225, E3 +366917.517}
SPL {X  -165.650, Y  +611.479, Z    +0.000, E1   +52.226, E3 +366931.069}
SPL {X  -165.650, Y  +599.923, Z    +0.000, E1   +51.240, E3 +366948.158}
SPL {X  -165.650, Y  +553.219, Z    +0.000, E1   +52.865, E3 +367004.919}
ENDSPLINE

SPLINE
SPL {X  -165.650, Y  +569.883, Z    +0.000, E1   +45.183, E3 +367020.596}
ENDSPLINE

SPLINE
SPL {X  -165.650, Y  +561.960, Z    +0.000, E1   +45.285, E3 +367036.251}
SPL {X  -165.650, Y  +554.065, Z    +0.000, E1   +45.254, E3 +367052.313}
SPL {X  -165.650, Y  +548.074, Z    +0.000, E1   +45.245, E3 +367064.424}
SPL {X  -165.650, Y  +542.958, Z    +0.000, E1   +45.131, E3 +367075.554}
SPL {X  -165.650, Y  +535.288, Z    +0.000, E1   +45.332, E3 +367089.995}
SPL {X  -165.650, Y  +529.160, Z    +0.000, E1   +45.215, E3 +367102.976}
SPL {X  -165.650, Y  +522.672, Z    +0.000, E1   +45.331, E3 +367115.542}
SPL {X  -165.650, Y  +516.211, Z    +0.000, E1   +45.175, E3 +367129.502}
SPL {X  -165.650, Y  +509.762, Z    +0.000, E1   +45.191, E3 +367142.544}
SPL {X  -165.650, Y  +503.812, Z    +0.000, E1   +45.188, E3 +367154.583}
SPL {X  -165.650, Y  +499.646, Z    +0.000, E1   +44.886, E3 +367164.854}
ENDSPLINE

SPLINE
SPL {X  -165.650, Y  +516.930, Z    +0.000, E1   +36.544, E3 +367173.524}
ENDSPLINE

SPLINE
SPL {X  -165.650, Y  +511.324, Z    +0.000, E1   +37.254, E3 +367184.515}
SPL {X  -165.650, Y  +504.742, Z    +0.000, E1   +38.087, E3 +367196.820}
SPL {X  -165.650, Y  +497.845, Z    +0.000, E1   +39.022, E3 +367208.895}
SPL {X  -165.650, Y  +491.819, Z    +0.000, E1   +39.756, E3 +367219.414}
SPL {X  -165.650, Y  +485.086, Z    +0.000, E1   +40.678, E3 +367230.258}
SPL {X  -165.650, Y  +476.633, Z    +0.000, E1   +41.847, E3 +367242.957}
SPL {X  -165.650, Y  +468.596, Z    +0.000, E1   +42.673, E3 +367256.220}
SPL {X  -165.650, Y  +460.562, Z    +0.000, E1   +43.733, E3 +367267.372}
SPL {X  -165.650, Y  +455.629, Z    +0.000, E1   +44.293, E3 +367274.491}
SPL {X  -165.650, Y  +449.099, Z    +0.000, E1   +44.871, E3 +367284.723}
SPL {X  -165.650, Y  +442.120, Z    +0.000, E1   +45.313, E3 +367296.275}
SPL {X  -165.650, Y  +439.103, Z    +0.000, E1   +44.726, E3 +367305.884}
SPL {X  -165.650, Y  +433.421, Z    +0.000, E1   +45.110, E3 +367315.272}
SPL {X  -165.650, Y  +426.476, Z    +0.000, E1   +45.244, E3 +367328.775}
SPL {X  -165.650, Y  +420.418, Z    +0.000, E1   +45.128, E3 +367341.569}
SPL {X  -165.650, Y  +415.564, Z    +0.000, E1   +45.195, E3 +367351.114}
SPL {X  -165.650, Y  +410.687, Z    +0.000, E1   +44.955, E3 +367362.430}
SPL {X  -165.650, Y  +402.778, Z    +0.000, E1   +45.323, E3 +367376.511}
SPL {X  -165.650, Y  +396.171, Z    +0.000, E1   +44.969, E3 +367391.932}
SPL {X  -165.650, Y  +390.060, Z    +0.000, E1   +45.007, E3 +367404.165}
SPL {X  -165.650, Y  +383.700, Z    +0.000, E1   +45.345, E3 +367415.089}
SPL {X  -165.650, Y  +379.225, Z    +0.000, E1   +45.073, E3 +367425.778}
SPL {X  -165.591, Y  +374.097, Z    +0.000, E1   +45.069, E3 +367436.259}
SPL {X  -165.372, Y  +368.914, Z    +0.000, E1   +45.103, E3 +367446.619}
SPL {X  -164.833, Y  +362.064, Z    +0.000, E1   +44.999, E3 +367461.404}
SPL {X  -164.024, Y  +355.348, Z    +0.000, E1   +45.002, E3 +367474.792}
SPL {X  -163.441, Y  +351.538, Z    +0.000, E1   +44.749, E3 +367484.008}
SPL {X  -162.419, Y  +345.942, Z    +0.000, E1   +44.540, E3 +367496.740}
SPL {X  -161.210, Y  +340.404, Z    +0.000, E1   +44.250, E3 +367509.565}
SPL {X  -159.961, Y  +335.460, Z    +0.000, E1   +44.205, E3 +367519.928}
SPL {X  -158.595, Y  +330.672, Z    +0.000, E1   +43.797, E3 +367531.906}
SPL {X  -156.695, Y  +324.773, Z    +0.000, E1   +43.987, E3 +367542.803}
SPL {X  -148.318, Y  +304.733, Z    +0.000, E1   +49.897, E3 +367548.039}
SPL {X  -138.435, Y  +287.529, Z    +0.000, E1   +45.834, E3 +367613.364}
SPL {X  -134.645, Y  +282.008, Z    +0.000, E1   +45.207, E3 +367643.020}
ENDSPLINE

SPLINE
SPL {X  -154.915, Y  +319.839, Z    +0.000, E1   +31.584, E3 +367702.539}
SPL {X  -161.387, Y  +341.161, Z    +0.000, E1   +22.590, E3 +367716.385}
SPL {X  -164.566, Y  +359.576, Z    +0.000, E1   +13.425, E3 +367694.978}
SPL {X  -165.355, Y  +368.611, Z    +0.000, E1    +8.407, E3 +367698.559}
SPL {X  -165.614, Y  +375.050, Z    +0.000, E1    +4.520, E3 +367699.863}
SPL {X  -165.650, Y  +379.847, Z    +0.000, E1    +1.364, E3 +367698.212}
SPL {X  -165.650, Y  +383.246, Z    +0.000, E1    -1.216, E3 +367697.306}
SPL {X  -165.650, Y  +386.866, Z    +0.000, E1    -4.337, E3 +367697.358}
SPL {X  -165.650, Y  +394.200, Z    +0.000, E1   -11.943, E3 +367695.125}
SPL {X  -165.650, Y  +405.401, Z    +0.000, E1   -24.512, E3 +367694.945}
SPL {X  -165.650, Y  +418.038, Z    +0.000, E1   -38.688, E3 +367691.173}
SPL {X  -165.650, Y  +461.620, Z    +0.000, E1   -55.594, E3 +367711.351}
SPL {X  -165.650, Y  +498.574, Z    +0.000, E1   -52.082, E3 +367772.377}
ENDSPLINE

SPLINE
SPL {X  -165.650, Y  +484.983, Z    +0.000, E1   -45.406, E3 +367787.879}
ENDSPLINE

SPLINE
SPL {X  -165.650, Y  +492.090, Z    +0.000, E1   -45.292, E3 +367802.902}
SPL {X  -165.650, Y  +498.857, Z    +0.000, E1   -45.339, E3 +367816.239}
SPL {X  -165.650, Y  +505.115, Z    +0.000, E1   -45.299, E3 +367829.187}
SPL {X  -165.650, Y  +510.931, Z    +0.000, E1   -45.250, E3 +367841.178}
SPL {X  -165.650, Y  +516.157, Z    +0.000, E1   -45.240, E3 +367851.852}
SPL {X  -165.650, Y  +521.049, Z    +0.000, E1   -45.236, E3 +367861.805}
SPL {X  -165.650, Y  +527.050, Z    +0.000, E1   -45.345, E3 +367873.301}
SPL {X  -165.650, Y  +532.042, Z    +0.000, E1   -45.233, E3 +367884.044}
SPL {X  -165.650, Y  +537.290, Z    +0.000, E1   -45.204, E3 +367894.885}
SPL {X  -165.650, Y  +544.196, Z    +0.000, E1   -45.432, E3 +367907.559}
SPL {X  -165.650, Y  +548.678, Z    +0.000, E1   -45.162, E3 +367918.123}
SPL {X  -165.650, Y  +554.600, Z    +0.000, E1   -45.345, E3 +367929.100}
SPL {X  -165.650, Y  +559.896, Z    +0.000, E1   -45.150, E3 +367940.956}
SPL {X  -165.650, Y  +566.830, Z    +0.000, E1   -45.346, E3 +367953.936}
SPL {X  -165.650, Y  +573.074, Z    +0.000, E1   -45.379, E3 +367966.267}
SPL {X  -165.650, Y  +579.360, Z    +0.000, E1   -45.300, E3 +367979.552}
SPL {X  -165.650, Y  +584.577, Z    +0.000, E1   -45.167, E3 +367990.775}
SPL {X  -165.650, Y  +590.060, Z    +0.000, E1   -45.221, E3 +368001.666}
SPL {X  -165.650, Y  +596.611, Z    +0.000, E1   -45.390, E3 +368013.902}
SPL {X  -165.650, Y  +603.637, Z    +0.000, E1   -45.296, E3 +368028.821}
SPL {X  -165.650, Y  +610.850, Z    +0.000, E1   -45.208, E3 +368043.829}
SPL {X  -165.650, Y  +617.450, Z    +0.000, E1   -45.402, E3 +368056.031}
SPL {X  -165.650, Y  +622.720, Z    +0.000, E1   -45.272, E3 +368067.429}
SPL {X  -165.650, Y  +627.828, Z    +0.000, E1   -45.174, E3 +368078.386}
SPL {X  -165.650, Y  +634.620, Z    +0.000, E1   -45.438, E3 +368090.592}
SPL {X  -165.650, Y  +640.808, Z    +0.000, E1   -45.294, E3 +368103.966}
SPL {X  -165.650, Y  +646.552, Z    +0.000, E1   -45.137, E3 +368116.490}
SPL {X  -165.650, Y  +652.431, Z    +0.000, E1   -45.333, E3 +368127.245}
SPL {X  -165.650, Y  +657.443, Z    +0.000, E1   -45.316, E3 +368137.501}
SPL {X  -165.650, Y  +662.999, Z    +0.000, E1   -45.214, E3 +368149.373}
SPL {X  -165.650, Y  +668.737, Z    +0.000, E1   -45.236, E3 +368160.888}
SPL {X  -165.650, Y  +675.226, Z    +0.000, E1   -45.503, E3 +368172.392}
SPL {X  -165.597, Y  +679.672, Z    +0.000, E1   -45.206, E3 +368183.113}
SPL {X  -165.388, Y  +684.808, Z    +0.000, E1   -45.192, E3 +368193.620}
SPL {X  -165.020, Y  +689.938, Z    +0.000, E1   -45.107, E3 +368204.563}
SPL {X  -164.358, Y  +696.147, Z    +0.000, E1   -45.160, E3 +368216.829}
SPL {X  -163.631, Y  +701.286, Z    +0.000, E1   -44.994, E3 +368228.121}
SPL {X  -162.679, Y  +706.734, Z    +0.000, E1   -44.812, E3 +368240.354}
SPL {X  -161.655, Y  +711.661, Z    +0.000, E1   -44.525, E3 +368251.735}
SPL {X  -160.692, Y  +715.726, Z    +0.000, E1   -44.379, E3 +368260.892}
SPL {X  -159.384, Y  +720.631, Z    +0.000, E1   -44.155, E3 +368272.042}
SPL {X  -158.321, Y  +724.227, Z    +0.000, E1   -43.955, E3 +368280.363}
SPL {X  -156.604, Y  +729.490, Z    +0.000, E1   -44.229, E3 +368289.530}
SPL {X  -147.100, Y  +751.668, Z    +0.000, E1   -50.624, E3 +368295.417}
SPL {X  -144.116, Y  +757.172, Z    +0.000, E1   -42.809, E3 +368364.813}
SPL {X  -127.227, Y  +781.582, Z    +0.000, E1   -46.780, E3 +368410.482}
ENDSPLINE

SPLINE
SPL {X  -133.736, Y  +773.248, Z    +0.000, E1   -45.385, E3 +368488.525}
SPL {X  -160.761, Y  +715.447, Z    +0.000, E1   -23.748, E3 +368445.375}
SPL {X  -164.304, Y  +696.571, Z    +0.000, E1   -14.525, E3 +368450.599}
SPL {X  -165.498, Y  +682.585, Z    +0.000, E1    -6.769, E3 +368450.273}
SPL {X  -165.650, Y  +674.975, Z    +0.000, E1    -1.888, E3 +368448.631}
SPL {X  -165.650, Y  +671.520, Z    +0.000, E1    +0.682, E3 +368447.559}
SPL {X  -165.650, Y  +668.289, Z    +0.000, E1    +3.417, E3 +368447.401}
SPL {X  -165.650, Y  +663.040, Z    +0.000, E1    +8.602, E3 +368446.595}
SPL {X  -165.650, Y  +655.692, Z    +0.000, E1   +17.061, E3 +368445.130}
SPL {X  -165.650, Y  +646.511, Z    +0.000, E1   +26.434, E3 +368447.911}
SPL {X  -165.650, Y  +637.905, Z    +0.000, E1   +40.225, E3 +368436.035}
SPL {X  -165.650, Y  +611.479, Z    +0.000, E1   +52.226, E3 +368449.588}
SPL {X  -165.650, Y  +599.923, Z    +0.000, E1   +51.240, E3 +368466.677}
SPL {X  -165.650, Y  +553.219, Z    +0.000, E1   +52.865, E3 +368523.437}
ENDSPLINE

SPLINE
SPL {X  -165.650, Y  +569.883, Z    +0.000, E1   +45.183, E3 +368539.114}
ENDSPLINE

SPLINE
SPL {X  -165.650, Y  +561.960, Z    +0.000, E1   +45.285, E3 +368554.769}
SPL {X  -165.650, Y  +554.065, Z    +0.000, E1   +45.254, E3 +368570.831}
SPL {X  -165.650, Y  +548.074, Z    +0.000, E1   +45.245, E3 +368582.942}
SPL {X  -165.650, Y  +542.958, Z    +0.000, E1   +45.131, E3 +368594.073}
SPL {X  -165.650, Y  +535.288, Z    +0.000, E1   +45.332, E3 +368608.514}
SPL {X  -165.650, Y  +529.160, Z    +0.000, E1   +45.215, E3 +368621.495}
SPL {X  -165.650, Y  +522.672, Z    +0.000, E1   +45.331, E3 +368634.061}
SPL {X  -165.650, Y  +516.211, Z    +0.000, E1   +45.175, E3 +368648.020}
SPL {X  -165.650, Y  +509.762, Z    +0.000, E1   +45.191, E3 +368661.062}
SPL {X  -165.650, Y  +503.812, Z    +0.000, E1   +45.188, E3 +368673.101}
SPL {X  -165.650, Y  +499.646, Z    +0.000, E1   +44.886, E3 +368683.372}
ENDSPLINE

SPLINE
SPL {X  -165.650, Y  +514.834, Z    +0.000, E1   +36.829, E3 +368696.138}
ENDSPLINE

SPLINE
SPL {X  -165.650, Y  +506.421, Z    +0.000, E1   +37.886, E3 +368712.250}
SPL {X  -165.650, Y  +499.917, Z    +0.000, E1   +38.752, E3 +368723.711}
SPL {X  -165.650, Y  +493.826, Z    +0.000, E1   +39.521, E3 +368734.465}
SPL {X  -165.650, Y  +487.003, Z    +0.000, E1   +40.380, E3 +368745.919}
SPL {X  -165.650, Y  +478.382, Z    +0.000, E1   +41.628, E3 +368758.832}
SPL {X  -165.650, Y  +472.112, Z    +0.000, E1   +42.202, E3 +368769.571}
SPL {X  -165.650, Y  +466.741, Z    +0.000, E1   +42.890, E3 +368777.491}
SPL {X  -165.650, Y  +458.202, Z    +0.000, E1   +44.020, E3 +368789.279}
SPL {X  -165.650, Y  +449.099, Z    +0.000, E1   +44.871, E3 +368803.242}
SPL {X  -165.650, Y  +442.120, Z    +0.000, E1   +45.313, E3 +368814.794}
SPL {X  -165.650, Y  +436.063, Z    +0.000, E1   +44.972, E3 +368829.378}
SPL {X  -165.650, Y  +427.943, Z    +0.000, E1   +45.362, E3 +368843.415}
SPL {X  -165.650, Y  +422.523, Z    +0.000, E1   +45.103, E3 +368856.094}
SPL {X  -165.650, Y  +415.564, Z    +0.000, E1   +45.195, E3 +368869.633}
SPL {X  -165.650, Y  +410.687, Z    +0.000, E1   +44.955, E3 +368880.949}
SPL {X  -165.650, Y  +405.522, Z    +0.000, E1   +45.119, E3 +368890.509}
SPL {X  -165.650, Y  +399.216, Z    +0.000, E1   +45.246, E3 +368902.703}
SPL {X  -165.650, Y  +391.618, Z    +0.000, E1   +45.037, E3 +368919.481}
SPL {X  -165.650, Y  +383.700, Z    +0.000, E1   +45.345, E3 +368933.607}
SPL {X  -165.650, Y  +379.225, Z    +0.000, E1   +45.073, E3 +368944.296}
SPL {X  -165.591, Y  +374.097, Z    +0.000, E1   +45.069, E3 +368954.777}
SPL {X  -165.372, Y  +368.914, Z    +0.000, E1   +45.103, E3 +368965.137}
SPL {X  -164.987, Y  +363.696, Z    +0.000, E1   +45.006, E3 +368976.360}
SPL {X  -164.256, Y  +357.053, Z    +0.000, E1   +44.969, E3 +368990.163}
SPL {X  -163.441, Y  +351.538, Z    +0.000, E1   +44.749, E3 +369002.527}
SPL {X  -162.419, Y  +345.942, Z    +0.000, E1   +44.540, E3 +369015.258}
SPL {X  -161.210, Y  +340.404, Z    +0.000, E1   +44.250, E3 +369028.083}
SPL {X  -159.961, Y  +335.460, Z    +0.000, E1   +44.205, E3 +369038.446}
SPL {X  -158.595, Y  +330.672, Z    +0.000, E1   +43.797, E3 +369050.424}
SPL {X  -156.695, Y  +324.773, Z    +0.000, E1   +43.987, E3 +369061.321}
SPL {X  -148.318, Y  +304.733, Z    +0.000, E1   +49.897, E3 +369066.558}
SPL {X  -138.435, Y  +287.529, Z    +0.000, E1   +45.834, E3 +369131.882}
SPL {X  -137.083, Y  +285.505, Z    +0.000, E1   +44.955, E3 +369150.047}
ENDSPLINE

SPLINE
SPL {X  -137.518, Y  +286.149, Z    +0.000, E1   +42.648, E3 +369213.927}
SPL {X  -156.430, Y  +324.005, Z    +0.000, E1   +29.926, E3 +369219.062}
SPL {X  -161.387, Y  +341.161, Z    +0.000, E1   +22.590, E3 +369234.903}
SPL {X  -164.566, Y  +359.576, Z    +0.000, E1   +13.425, E3 +369213.497}
SPL {X  -165.355, Y  +368.611, Z    +0.000, E1    +8.407, E3 +369217.078}
SPL {X  -165.614, Y  +375.050, Z    +0.000, E1    +4.520, E3 +369218.381}
SPL {X  -165.650, Y  +379.847, Z    +0.000, E1    +1.364, E3 +369216.731}
SPL {X  -165.650, Y  +383.246, Z    +0.000, E1    -1.216, E3 +369215.824}
SPL {X  -165.650, Y  +386.866, Z    +0.000, E1    -4.337, E3 +369215.877}
SPL {X  -165.650, Y  +394.200, Z    +0.000, E1   -11.943, E3 +369213.644}
SPL {X  -165.650, Y  +405.401, Z    +0.000, E1   -24.512, E3 +369213.464}
SPL {X  -165.650, Y  +418.038, Z    +0.000, E1   -38.688, E3 +369209.691}
SPL {X  -165.650, Y  +461.620, Z    +0.000, E1   -55.594, E3 +369229.870}
SPL {X  -165.650, Y  +498.574, Z    +0.000, E1   -52.082, E3 +369290.895}
ENDSPLINE

SPLINE
SPL {X  -165.650, Y  +484.983, Z    +0.000, E1   -45.406, E3 +369306.398}
ENDSPLINE

